   If rst303.EOF = False Then
   	SmartTags("ID_OP_4") = rst303.Fields(0).Value
   	SmartTags("Name_OP_4") = rst303.Fields(1).Value
   	rst303.MoveNext
   Else
   	SmartTags("ID_OP_4") = 0
   	SmartTags("Name_OP_4") = "Vacio"
   End If
   
   If rst303.EOF = False Then
   	SmartTags("ID_OP_5") = rst303.Fields(0).Value
   	SmartTags("Name_OP_5") = rst303.Fields(1).Value
   	rst303.MoveNext
   Else
   	SmartTags("ID_OP_5") = 0
   	SmartTags("Name_OP_5") = "Vacio"
   End If
   
   rst303.close
   conn303.close
   
   Set rst303 = Nothing
   Set conn303 = Nothing

VB script "S20_Generador_Inf"
   Dim NombreInf_Pl, NombreInf_Lavs
   
   'Informe de planchadoras
   bfde4b54-0db7-4817-8032-87127bf19bb9 "Se llamo a S07"
   NombreInf_Pl = S07_InformeDiario_Planchas()
   bfde4b54-0db7-4817-8032-87127bf19bb9 "Se Salio de S07"
   
   ' Informe unico de lavadoras
   bfde4b54-0db7-4817-8032-87127bf19bb9 "Se llamo a S23"
   NombreInf_Lavs = S23_Creador_InformeDiarioLavs_Gral()
   bfde4b54-0db7-4817-8032-87127bf19bb9 "Se Salio de S23"
   
   Call S30_EnvioInformes_Email(NombreInf_Pl, NombreInf_Lavs)

VB script "S30_EnvioInformes_Email"
   '## ENVIAR INFORME POR EMAIL
   
   Dim appOutlook 'As OUTLOOK.APPLICATION
   Dim mlNewMail 'As MailItem
   Dim objEntry
   Dim Text
   
   Const addressee = "crj@eprocsrl.com.ar; danielst@live.com.ar; josemariacullen@hotmail.com;"' zekeserio@hotmail.com;"
   
   ' Text to be sent 
   
   Text = "Informe diario"
   
   Set appOutlook = CreateObject("OUTLOOK.APPLICATION")
   
   
   'Generating and sending an e-mail:
   Set mlNewMail = appOutlook.CreateItem(0)
   mlNewMail.Display
   mlNewMail.To = addressee
   mlNewMail.Subject = "Informe Diario de produccion"
   
   
   If InStr(Arch1,"ERR") <> 0 Then
   	Text = Text + vbCrLf +_
   	"Error al Crear el informe de Planchadoras"
   Else
   	mlNewMail.Attachments.Add CStr(Arch1)
   End If
   
   If InStr(Arch2,"ERR") <> 0 Then
   	Text = Text + vbCrLf +_
   	"Error al Crear el informe de Lavadoras"
   Else
   	mlNewMail.Attachments.Add CStr(Arch2)
   End If
   
   
   mlNewMail.Body = Text
   mlNewMail.save
   mlNewMail.send 
   
   'Error routine
   If Err.Number <> 0 Then
   	bfde4b54-0db7-4817-8032-87127bf19bb9 "Error al enviar el email #" & Err.Number & " " & Err.Description
   End If

VB script "S304_ActualizarOpEnPrincipal"
   'Declaracion de Variables locales
   Dim conn21, rst21, Consulta
   
   On Error Resume Next
   
   Set conn21 = CreateObject("ADODB.Connection")
   Set rst21 = CreateObject("ADODB.Recordset")
   
   'Abrir BDD
   conn21.Open "Provider=MSDASQL;Initial Catalog=Lavadero;DSN=Lavadero"
   
   
   'Chequeo de error
   If Err.Number <> 0 Then
   	bfde4b54-0db7-4817-8032-87127bf19bb9 "Error #" & Err.Number & " " & Err.Description
   	Err.Clear 
   	Set conn21 = Nothing
   	Exit Sub
   End If
   
   If LavNro = 1 Then	
   	
   	Consulta = "SELECT * FROM Op_Lavadoras WHERE  ID = '" & SmartTags("Lav1_Operador") &"';"
   	
   	'Ejecutar consulta
   	Set rst21 = conn21.Execute(Consulta)
   
   	SmartTags("Lav1_Operador_Str")= rst21.Fields(1).Value
   	
   End If
   
   If LavNro = 2 Then	
   	Consulta = "SELECT * FROM Op_Lavadoras WHERE  ID = '" & SmartTags("Lav2_Operador") &"';"
   	
   	'Ejecutar consulta
   	Set rst21 = conn21.Execute(Consulta)
   
   	SmartTags("Lav2_Operador_Str")= rst21.Fields(1).Value
   	
   End If
   
   If LavNro = 3 Then	
   	Consulta = "SELECT * FROM Op_Lavadoras WHERE  ID = '" & SmartTags("Lav3_Operador") &"';"
   	
   	'Ejecutar consulta
   	Set rst21 = conn21.Execute(Consulta)
   
   	SmartTags("Lav3_Operador_Str")= rst21.Fields(1).Value
   	
   End If
   
   If LavNro = 4 Then	
   	Consulta = "SELECT * FROM Op_Lavadoras WHERE  ID = '" & SmartTags("Lav4_Operador") &"';"
   	
   	'Ejecutar consulta
   	Set rst21 = conn21.Execute(Consulta)
   
   	SmartTags("Lav4_Operador_Str")= rst21.Fields(1).Value
   	
   End If
   
   
   rst21.close 
   
   conn21.close
   
   Set rst21 = Nothing
   Set conn21 = Nothing

VB script "SA1_email_Vibr"
   	
   	
   	Dim appOutlook 'As OUTLOOK.APPLICATION
   	Dim mlNewMail 'As MailItem
   	Dim objEntry
   	Dim Text, cliente_0, cliente_1, cliente_2, operario, carga, programa
   	Dim cliente_0_str, cliente_1_str, cliente_2_str, operario_str
   		
   	Const addressee = "crj@eprocsrl.com.ar; danielst@live.com.ar;"' josemariacullen@hotmail.com; zekeserio@hotmail.com;"	
   	
   	
   ' ######### Consulta para obtener el listado actualizado de clientes ############
   	Dim conncli, rstcli , ConsultaCli
   	
   	Set conncli = CreateObject("ADODB.Connection")
   	Set rstcli = CreateObject("ADODB.Recordset")
   	
   	'Open data source - Datenquelle öffnen
   	conncli.Open "Provider=MSDASQL;Initial Catalog=Lavadero;DSN=Lavadero"
   	'Error routine - Fehlerroutine
   	If Err.Number <> 0 Then
   		bfde4b54-0db7-4817-8032-87127bf19bb9 "Conexion Error a Cli_Lavadoras#" & Err.Number & " " & Err.Description
   		Err.Clear
   		Set conncli = Nothing  
   		Exit Sub
   	End If
   	
   	ConsultaCli = "SELECT * FROM Cli_Lavadoras;"
   	
   	'Ejecutar consulta
   	Set rstcli = conncli.Execute(ConsultaCli)
   '''''''''''''''''''''''''''''''''''''''''''''''''''''''''''''''''''''''
   
   	
   ' ######### Consulta para obtener el listado actualizado de OPERADORES ############
   Dim connope, rstope , Consultaope
   
   Set connope = CreateObject("ADODB.Connection")
   Set rstope = CreateObject("ADODB.Recordset")
   
   'Open data source - Datenquelle öffnen
   connope.Open "Provider=MSDASQL;Initial Catalog=Lavadero;DSN=Lavadero"
   'Error routine - Fehlerroutine
   If Err.Number <> 0 Then
   	bfde4b54-0db7-4817-8032-87127bf19bb9 "Conexion Error a Op_Lavadoras" & Err.Number & " " & Err.Description
   	Err.Clear
   	Set connope = Nothing  
   	Exit Sub
   End If
   
   Consultaope = "SELECT * FROM Op_Lavadoras;"
   
   'Ejecutar consulta
   Set rstope = connope.Execute(Consultaope)
   ''''''''''''''''''''''''''''''''''''''''''''''''''''''''''''''''''''''''''''''''
   	
   '## ENVIAR Aviso POR EMAIL AVISO FALLA VIBRACION LAVADORA 1
   
   If  SmartTags("Lav1_AlarmaVibracion") = True Then
   
   	cliente_0 = SmartTags("Lav1_Cliente_0")
   	cliente_1 = SmartTags("Lav1_Cliente_1")
   	cliente_2 = SmartTags("Lav1_Cliente_2")
   		
   	operario = SmartTags("Lav1_Operador")
   	
   	carga = SmartTags("Lav1_CantRopa")
   	
   	programa =  S12_Conversor_BCD_to_Int(SmartTags("Lav1_Programa"))
   	
   
   	' Establecer los clientes
   	Do While rstcli.EOF = False
   		If (rstcli.Fields(0).Value = cliente_0) Then 
   			cliente_0_str = Trim(rstcli.Fields(1).Value)
   		End If
   
   		If (rstcli.Fields(0).Value = cliente_1) Then 
   			cliente_1_str = Trim(rstcli.Fields(1).Value)
   		End If
   
   		If (rstcli.Fields(0).Value = cliente_2) Then 
   			cliente_2_str = Trim(rstcli.Fields(1).Value)
   		End If
   			
   		rstcli.MoveNext
   	Loop
   	
   	' Establecer operador
   	Do While rstope.EOF = False
   		If (rstope.Fields(0).Value = operario) Then 
   			operario_str = Trim(rstope.Fields(1).Value)
   		End If	
   		rstope.MoveNext
   	Loop
   		
   	' Text to be sent 
   	
   	Text = "AVISO DE FALLA POR VIBRACION EN LAVADORA 1" + vbCrLf +_
   			"Hora: " + CStr(Date()) + " " + CStr(Time()) + vbCrLf +_
   			"Clientes: " + cliente_0_str + "/" + cliente_1_str + "/" + cliente_2_str + vbCrLf +_
   			"Operario: " + operario_str + vbCrLf +_
   			"Carga: " + CStr(carga/10) + " Kg" + vbCrLf +_
   			"Programa: " + CStr(programa)
   	
   	Set appOutlook = CreateObject("OUTLOOK.APPLICATION")
   	
   	
   	'Generating and sending an e-mail:
   	Set mlNewMail = appOutlook.CreateItem(0)
   	mlNewMail.Display
   	mlNewMail.To = addressee
   	mlNewMail.Subject = "Aviso de falla por vibracion en lavadora 1"
   	mlNewMail.Body = Text
   	mlNewMail.save
   	mlNewMail.send 
   	
   End If
   
   '## ENVIAR Aviso POR EMAIL AVISO FALLA VIBRACION LAVADORA 2
   
   If  SmartTags("Lav2_AlarmaVibracion") = True Then
   
   	cliente_0 = SmartTags("Lav2_Cliente_0")
   	cliente_1 = SmartTags("Lav2_Cliente_1")
   	cliente_2 = SmartTags("Lav2_Cliente_2")
   		
   	operario = SmartTags("Lav2_Operador")
   	
   	carga = SmartTags("Lav2_CantRopa")
   	
   	programa =  S12_Conversor_BCD_to_Int(SmartTags("Lav2_Programa"))
   	
   
   	' Establecer los clientes
   	Do While rstcli.EOF = False
   		If (rstcli.Fields(0).Value = cliente_0) Then 
   			cliente_0_str = Trim(rstcli.Fields(1).Value)
   		End If
   
   		If (rstcli.Fields(0).Value = cliente_1) Then 
   			cliente_1_str = Trim(rstcli.Fields(1).Value)
   		End If
   
   		If (rstcli.Fields(0).Value = cliente_2) Then 
   			cliente_2_str = Trim(rstcli.Fields(1).Value)
   		End If
   			
   		rstcli.MoveNext
   	Loop
   	
   	' Establecer operador
   	Do While rstope.EOF = False
   		If (rstope.Fields(0).Value = operario) Then 
   			operario_str = Trim(rstope.Fields(1).Value)
   		End If	
   		rstope.MoveNext
   	Loop
   		
   	' Text to be sent 
   	
   	Text = "AVISO DE FALLA POR VIBRACION EN LAVADORA 2" + vbCrLf +_
   			"Hora: " + CStr(Date()) + " " + CStr(Time()) + vbCrLf +_
   			"Clientes: " + cliente_0_str + "/" + cliente_1_str + "/" + cliente_2_str + vbCrLf +_
   			"Operario: " + operario_str + vbCrLf +_
   			"Carga: " + CStr(carga/10) + " Kg" + vbCrLf +_
   			"Programa: " + CStr(programa)
   	
   	Set appOutlook = CreateObject("OUTLOOK.APPLICATION")
   	
   	
   	'Generating and sending an e-mail:
   	Set mlNewMail = appOutlook.CreateItem(0)
   	mlNewMail.Display
   	mlNewMail.To = addressee
   	mlNewMail.Subject = "Aviso de falla por vibracion en lavadora 2"
   	mlNewMail.Body = Text
   	mlNewMail.save
   	mlNewMail.send 
   	
   End If
   
   '## ENVIAR Aviso POR EMAIL AVISO FALLA VIBRACION LAVADORA 3
   
   If  SmartTags("Lav3_AlarmaVibracion") = True Then
   
   	cliente_0 = SmartTags("Lav3_Cliente_0")
   	cliente_1 = SmartTags("Lav3_Cliente_1")
   	cliente_2 = SmartTags("Lav3_Cliente_2")
   		
   	operario = SmartTags("Lav3_Operador")
   	
   	carga = SmartTags("Lav3_CantRopa")
   	
   	programa =  S12_Conversor_BCD_to_Int(SmartTags("Lav3_Programa"))
   	
   
   	' Establecer los clientes
   	Do While rstcli.EOF = False
   		If (rstcli.Fields(0).Value = cliente_0) Then 
   			cliente_0_str = Trim(rstcli.Fields(1).Value)
   		End If
   
   		If (rstcli.Fields(0).Value = cliente_1) Then 
   			cliente_1_str = Trim(rstcli.Fields(1).Value)
   		End If
   
   		If (rstcli.Fields(0).Value = cliente_2) Then 
   			cliente_2_str = Trim(rstcli.Fields(1).Value)
   		End If
   			
   		rstcli.MoveNext
   	Loop
   	
   	' Establecer operador
   	Do While rstope.EOF = False
   		If (rstope.Fields(0).Value = operario) Then 
   			operario_str = Trim(rstope.Fields(1).Value)
   		End If	
   		rstope.MoveNext
   	Loop
   		
   	' Text to be sent 
   	
   	Text = "AVISO DE FALLA POR VIBRACION EN LAVADORA 3" + vbCrLf +_
   			"Hora: " + CStr(Date()) + " " + CStr(Time()) + vbCrLf +_
   			"Clientes: " + cliente_0_str + "/" + cliente_1_str + "/" + cliente_2_str + vbCrLf +_
   			"Operario: " + operario_str + vbCrLf +_
   			"Carga: " + CStr(carga/10) + " Kg" + vbCrLf +_
   			"Programa: " + CStr(programa)
   	
   	Set appOutlook = CreateObject("OUTLOOK.APPLICATION")
   	
   	
   	'Generating and sending an e-mail:
   	Set mlNewMail = appOutlook.CreateItem(0)
   	mlNewMail.Display
   	mlNewMail.To = addressee
   	mlNewMail.Subject = "Aviso de falla por vibracion en lavadora 3"
   	mlNewMail.Body = Text
   	mlNewMail.save
   	mlNewMail.send 
   	
   End If
   
   
   '## ENVIAR Aviso POR EMAIL AVISO FALLA VIBRACION LAVADORA 3
   
   If  SmartTags("Lav4_AlarmaVibracion") = True Then
   
   	cliente_0 = SmartTags("Lav4_Cliente_0")
   	cliente_1 = SmartTags("Lav4_Cliente_1")
   	cliente_2 = SmartTags("Lav4_Cliente_2")
   		
   	operario = SmartTags("Lav4_Operador")
   	
   	carga = SmartTags("Lav4_CantRopa")
   	
   	programa =  S12_Conversor_BCD_to_Int(SmartTags("Lav4_Programa"))
   	
   
   	' Establecer los clientes
   	Do While rstcli.EOF = False
   		If (rstcli.Fields(0).Value = cliente_0) Then 
   			cliente_0_str = Trim(rstcli.Fields(1).Value)
   		End If
   
   		If (rstcli.Fields(0).Value = cliente_1) Then 
   			cliente_1_str = Trim(rstcli.Fields(1).Value)
   		End If
   
   		If (rstcli.Fields(0).Value = cliente_2) Then 
   			cliente_2_str = Trim(rstcli.Fields(1).Value)
   		End If
   			
   		rstcli.MoveNext
   	Loop
   	
   	' Establecer operador
   	Do While rstope.EOF = False
   		If (rstope.Fields(0).Value = operario) Then 
   			operario_str = Trim(rstope.Fields(1).Value)
   		End If	
   		rstope.MoveNext
   	Loop
   		
   	' Text to be sent 
   	
   	Text = "AVISO DE FALLA POR VIBRACION EN LAVADORA 4" + vbCrLf +_
   			"Hora: " + CStr(Date()) + " " + CStr(Time()) + vbCrLf +_
   			"Clientes: " + cliente_0_str + "/" + cliente_1_str + "/" + cliente_2_str + vbCrLf +_
   			"Operario: " + operario_str + vbCrLf +_
   			"Carga: " + CStr(carga/10) + " Kg" + vbCrLf +_
   			"Programa: " + CStr(programa)
   	
   	Set appOutlook = CreateObject("OUTLOOK.APPLICATION")
   	
   	
   	'Generating and sending an e-mail:
   	Set mlNewMail = appOutlook.CreateItem(0)
   	mlNewMail.Display
   	mlNewMail.To = addressee
   	mlNewMail.Subject = "Aviso de falla por vibracion en lavadora 4"
   	mlNewMail.Body = Text
   	mlNewMail.save
   	mlNewMail.send 
   	
   End If
   
   
   
   '########################################################################
   'Close data source - Datenquelle schließen
   
   conncli.close
   Set rstcli = Nothing
   Set conncli = Nothing
   
   connope.close
   Set rstope = Nothing
   Set connope = Nothing

VB script "S23_Creador_InformeDiarioLavs_Gral"
   S23_Creador_InformeDiarioLavs_Gral = "ERROR"
   
   If Err.Number <> 0 Then
   	bfde4b54-0db7-4817-8032-87127bf19bb9 "Erorr anterior a  'S23_Creador_InformeDiarioLavs_Gral' #" & Err.Number & " " & Err.Description
   	Err.Clear
   End If
   
   bfde4b54-0db7-4817-8032-87127bf19bb9 "Entro a S23"
   'Declaration of local tags 
   
   Dim cantidadDeRegistros
   	cantidadDeRegistros = 60
   Dim cantidadDeLavadoras
   	cantidadDeLavadoras = 4
   
   Dim conn, rst, i, j, indicehoja, k, l
   
   Dim Consulta
   Dim conncli, rstcli , ConsultaCli
   Dim connope, rstope , Consultaope
   Dim connfall,rstfall, Consultafall
   
   Dim DiaAnterior
   Dim horaInicioDia, horaFinDia
   Dim tcargaLav(4), tciclosLav(4), tciclosnvLav(4)
   Dim HoraFin, HoraInicio
   Dim thoras , tcarga, tciclos, thorasdate, thorasSdate(4), thorasmuertodate
   Dim rst2
   
   ' Creo Variables locales para poder iterar con los datos
   Dim VarCLINro_0(60), 	VarCLINro_1(60)
   Dim VarCLINro_2(60), 	VarC(60)
   Dim VarPR(60), 		VarHI(60)
   Dim VarHF(60), 		VarOPNro(60)
   Dim VarNV(60), 		VarEsp(60)
   Dim VarCLIStr(60), 	VarOPStr(60)
   Dim band_1(60), 	VarHE(60)
   Dim VarCicloOk(60), VarFalla(60), VarCicloOkAns(60)
   Dim VarCicloOk_CN(60)
   Dim VarFallaStr(60), VarFallaSQL(60)
   Dim LavadoraNro
   Dim indexMuertoFin(4),indexMuerto(4)
   Dim inicioderegistrosdelavadora
   Dim Programas(15), p, Promedio(4), PromedioTotal, Programas_Lav4(15)
   Dim fin
   Dim tiemponulo , thorasAns, tdias
   Dim lavEnFalla
   
   'Inicializacion Global de variables
   For p = 1 To 15
   	Programas(p) = 0
   	Programas_Lav4(p) = 0
   Next
   '
   If Err.Number <> 0 Then
   	bfde4b54-0db7-4817-8032-87127bf19bb9 "Consulta Lav Error 1#" & Err.Number & " " & Err.Description
   	Err.Clear
   	'Close data source	
   	Set conn = Nothing
   	Set rst = Nothing 
   	
   	Exit Function
   End If
   
   tiemponulo = FormatDateTime("2020-02-05 00:00:00", 4)
   
   For i = 1 To cantidadDeRegistros
   	VarNV(i) 		= 0
   	VarHI(i) 		= FormatDateTime("2020-02-05 00:00:00", 4)
   	VarHF(i) 		= FormatDateTime("2020-02-05 00:00:00", 4)
   	VarHE(i) 		= FormatDateTime("2020-02-05 00:00:00", 4)		
   	VarCLIStr(i) 	= "                                       "
   	VarOPStr(i) 	= "                                       "
   	band_1(i)		= 0
   	VarCicloOk(i)	= "X" ' negativo "O"; positivo "P"
   	VarFalla(i)		= 0
   	VarFallaStr(i)	= "                                       "	
   Next
   
   
   
   If Err.Number <> 0 Then
   	bfde4b54-0db7-4817-8032-87127bf19bb9 "Consulta Lav Error 2#" & Err.Number & " " & Err.Description
   	Err.Clear
   	'Close data source
   	Set conn = Nothing
   	Set rst = Nothing 
   	
   	Exit Function
   End If
   
   thoras = FormatDateTime("2020-02-05 00:00:00", 4)
   
   indicehoja = 1
   
   'DiaAnterior = Date() ' Es el día actual
   'DiaAnterior = DateAdd("d",-1, DiaAnterior)
   DiaAnterior = FormatDateTime(CStr(SmartTags("Ver_DIA_X")), 2)
   
   
   If Err.Number <> 0 Then
   	bfde4b54-0db7-4817-8032-87127bf19bb9 "Consulta Lav Error 3#" & Err.Number & " " & Err.Description
   	Err.Clear
   	'Close data source
   	Set conn = Nothing
   	Set rst = Nothing 
   	Exit Function
   End If
   
   
   For i = 1 To cantidadDeLavadoras
   	tcargaLav(i)		= 0
   	tciclosLav(i)		= 0
   	tciclosnvLav(i) 	= 0
   
   	Promedio(i)			= 0
   Next
   
   If Err.Number <> 0 Then
   	bfde4b54-0db7-4817-8032-87127bf19bb9 "Consulta Lav Error 5#" & Err.Number & " " & Err.Description
   	Err.Clear
   	'Close data source
   	Set conn = Nothing
   	Set rst = Nothing 
   	
   	Exit Function
   End If
   
   tcarga 			= 0
   tciclos 		= 0
   lavEnFalla		= 1
   
   'Analisar si hay error e imprimirlo
   If Err.Number <> 0 Then
   	bfde4b54-0db7-4817-8032-87127bf19bb9 "Consulta Lav Error 6#" & Err.Number & " " & Err.Description
   	Err.Clear
   	'Close data source
   	Set conn = Nothing
   	Set rst = Nothing 
   	
   	Exit Function
   End If
   
   ' Comienzo de procesamiento de datos
   On Error Resume Next
   
   For LavadoraNro = 1 To cantidadDeLavadoras
   	'""""""""""""""""""""""""""""""""""""""""""""""""""""""""""""""""""""""""""""""""""""
   	' #################   Generacion de consulta a BDD Lavadora   ######################
   	'------------------------------------------------------------------------------------
   	'############ Estructura de datos de la Tabla Lav1 #################################
   	
   	'0			1			2			3			4			5			6			7			8			
   	'|FechaFin	|FechIni	|Cliente_0	|Cliente_1	|Cliente_2	|Operario	|Carga		|Programa	|Valido
   	'|Date		|Date		|Int		|Int		|Int		|Int		|Int 100g	|Int		|Bool
   	
   	'##################################################################################
   		
   	'''''''''''''''''''''''''''''''''''''''''''''''''''''''''''''''''''''''''''''
   	' #################   Procesamieno de Datos   #############################
   	'----------------------------------------------------------------------------
   	
   	'Ejecutar consulta
   	
   	Consulta = "SELECT * FROM Lav" & LavadoraNro & " WHERE cast(fechafin As Date) = '"
   	Consulta = Consulta & CStr(Year(DiaAnterior)) & "-" & CStr(Month(DiaAnterior)) & "-" & CStr(Day(DiaAnterior)) & "' "
   	Consulta = Consulta & " order by fechafin"
   	
   	Set conn = CreateObject("ADODB.Connection")
   	conn.Open "Provider=MSDASQL;Initial Catalog=Lavadero;DSN=Lavadero"
   	Set rst2 = CreateObject("ADODB.Recordset")
   	Set rst2 = conn.Execute(Consulta)	
   	
   	inicioderegistrosdelavadora = indicehoja
   	i = indicehoja
   	
   	'ShowSystemAlarm "Entra al loop de Lectura de registros de Lav nro " & LavadoraNro
   	
   	Do While rst2.EOF = False
   			
   		VarCLINro_0(i) 	= rst2.Fields(2).Value
   		VarCLINro_1(i) 	= rst2.Fields(3).Value
   		VarCLINro_2(i) 	= rst2.Fields(4).Value
   		VarC(i) 		= rst2.Fields(6).Value / 10
   		VarPR(i) 		= rst2.Fields(7).Value
   		VarHI(i) 		= FormatDateTime(CStr(rst2.Fields(1).Value), 4) 'Devuelve la parte Time de la fecha
   		VarHF(i) 		= FormatDateTime(CStr(rst2.Fields(0).Value), 4)
   		VarOPNro(i)		= rst2.Fields(5).Value
   		VarNV(i) 		= 1	
   		VarCicloOk_CN(i)= rst2.Fields(9).Value
   		
   		If rst2.Fields(8).Value = 0 Then ' Si el ciclo es no valido
   			If VarCicloOk_CN(i) = 0 Then
   				VarCicloOk(i) 			= "O" ' negativo "O"; positivo "P"
   			Else
   				VarCicloOk(i) 			= "8" ' negativo "O"; positivo "P"
   			End If
   			tciclosnvLav(LavadoraNro) = tciclosnvLav(LavadoraNro) +1
   		Else
   			VarCicloOk(i) 			= "P" ' negativo "O"; positivo "P"
   			If VarPR(i) <> 12 And VarPR(i) <> 11 Then
   				tciclosLav(LavadoraNro) = tciclosLav(LavadoraNro) 	+ 1
   			End If
   			'tcargaLav(LavadoraNro)	= tcargaLav(LavadoraNro) 	+ VarC(i)
   				
   				' Suma de formulas utilizadas
   			If LavadoraNro <> 4 Then
   				Programas(VarPR(i)) = Programas(VarPR(i)) + 1
   			Else
   				Programas_Lav4(VarPR(i)) = Programas_Lav4(VarPR(i)) + 1
   			End If
   			
   		End If
   		
   		'Suma de Carga lavada
   		If i > 1 Then
   			If VarCicloOk(i) = "P" And VarPR(i) <> 12 And VarPR(i) <> 11 Or (VarCicloOkAns(i) = "O" And (VarPR(i) = 12 Or VarPR(i) = 11)) Then
   				tcargaLav(LavadoraNro)	= tcargaLav(LavadoraNro) 	+ VarC(i)
   			End If
   		Else
   			If VarCicloOk(i) = "P" And VarPR(i) <> 12 And VarPR(i) <> 11 Then
   				tcargaLav(LavadoraNro)	= tcargaLav(LavadoraNro) 	+ VarC(i)
   			End If
   		End If
   		
   	
   		'Calculo de tiempo muerto si corresponde
   		If i > 1 Then'VarHI(i-1) <> tiemponulo Then
   			VarHE(i-1) = DateAdd("h", Hour(VarHI(i)) - Hour(VarHF(i-1)), VarHE(i-1))
   			VarHE(i-1) = DateAdd("n", Minute(VarHI(i)) - Minute(VarHF(i-1)), VarHE(i-1))				
   			VarHE(i-1) = DateAdd("s", Second(VarHI(i)) - Second(VarHF(i-1)), VarHE(i-1))
   		End If
   		
   		thoras = DateAdd("h", Hour(VarHF(i)) - Hour(VarHI(i)), thoras)
   		thoras = DateAdd("n", Minute(VarHF(i)) - Minute(VarHI(i)), thoras)
   		thoras = DateAdd("s", Second(VarHF(i)) - Second(VarHI(i)), thoras)
   		
   		If Hour(thoras) < Hour(thorasAns) Then
   			tdias = tdias + 1 
   			thorasAns = thoras
   		Else
   			thorasAns = thoras
   		End If
   		
   		If i > 1 Then
   			VarCicloOkAns(i) = VarCicloOk(i)
   		End If
   		
   		'Indice de lavados		
   		i = i + 1
   		
   		
   		rst2.MoveNext
   		
   		If Err.Number <> 0 Then
   			bfde4b54-0db7-4817-8032-87127bf19bb9 "Error en la asignacion de variables locales en loop#" & Err.Number & " " & Err.Description
   			Err.Clear
   			Set conn = Nothing  
   			Exit Function
   		End If
   	Loop
   	
   	'ShowSystemAlarm "Sale del loop de Lectura de registros de Lav nro " & LavadoraNro
   	
   	If Err.Number <> 0 Then
   		bfde4b54-0db7-4817-8032-87127bf19bb9 "Error en la asignacion de variables locales luego del loop#" & Err.Number & " " & Err.Description
   		Err.Clear
   		Set conn = Nothing  
   		Exit Function
   	End If
   	
   	VarCicloOk(i) 	= "P" ' negativo "O"; positivo "P"
   	VarC(i) 		= tcargaLav(LavadoraNro)
   	VarNV(i) 		= 1
   	
   	'''	
   	VarCLIStr		(i)	= "Total Lav Maq " & CStr(LavadoraNro)
   	VarPR			(i)	= 0
   	VarHI			(i)	= 0	
   	VarHF			(i)	= 0
   	VarOPStr		(i) = " "
   	VarFallaStr		(i)	= " "
   	VarHE			(i) = 0
   	''''
   	indicehoja = i + 1
   	
   	'Indice para sumar tiempos muertos
   	indexMuertoFin(LavadoraNro) 	= i - 1
   	indexMuerto(LavadoraNro)		= i - 2
   	SmartTags("BCDtoInt")			= indexMuerto(LavadoraNro)
   	SmartTags("BCDtoInt_Entrada")	= inicioderegistrosdelavadora
   	
   	'Calculo de tiempos muertos parciales de lavadoras
   	k = inicioderegistrosdelavadora
   
   	fin = False
   	
   	'ShowSystemAlarm "Entra al loop de suma de tiempos muertos de lav  " & LavadoraNro
   		
   	Do While fin = False
   		VarHE(indexMuertoFin(LavadoraNro)) = DateAdd("h",Hour(VarHE(k)), VarHE(indexMuertoFin(LavadoraNro)))
   		VarHE(indexMuertoFin(LavadoraNro)) = DateAdd("n",Minute(VarHE(k)), VarHE(indexMuertoFin(LavadoraNro)))			
   		VarHE(indexMuertoFin(LavadoraNro)) = DateAdd("s",Second(VarHE(k)), VarHE(indexMuertoFin(LavadoraNro)))
   		
   		If (k < indexMuerto(LavadoraNro)) Then
   			k = k + 1
   		Else
   			fin = True
   		End If
   	Loop
   	
   	'ShowSystemAlarm "Sale del loop de suma de tiempos muertos de lav  " & LavadoraNro
   	
   	If Err.Number <> 0 Then
   		bfde4b54-0db7-4817-8032-87127bf19bb9 "Error en la asignacion de variables locales a lo ultimo#" & Err.Number & " " & Err.Description
   		Err.Clear
   		Set conn = Nothing  
   		Exit Function
   	End If
   	
   	
   	conn.close
   	Set rst2 = Nothing
   	Set conn = Nothing
   	
   Next
   
   'ShowSystemAlarm "Sale del loop general de rst"
   
   'Armado de tiempo total de lavado
   Dim tHorasString
   tHorasString = SA2_TotalTimeToString(tdias, thoras)
   
   'calculo de tiempo muerto total y promedios de las 4 lavadoras
   Dim indiceFinal
   indiceFinal = indexMuertoFin(4) +2
   'ShowSystemAlarm "entra loop Promedio, Var E"
   For k = 1 To 4
   	
   	VarHE(indiceFinal) = DateAdd("h",Hour(VarHE(indexMuertoFin(k))), VarHE(indiceFinal))
   	VarHE(indiceFinal) = DateAdd("n",Minute(VarHE(indexMuertoFin(k))), VarHE(indiceFinal))				
   	VarHE(indiceFinal) = DateAdd("s",Second(VarHE(indexMuertoFin(k))), VarHE(indiceFinal))
   	
   	If tciclosLav(k) <> 0 Then
   		Promedio(k) = tcargaLav(k) / tciclosLav(k)	
   	End If
   Next
   'ShowSystemAlarm "Sale loop Promedio, Var E"
   
   VarNV			(indiceFinal) 	= 1
   	
   If Err.Number <> 0 Then
   	bfde4b54-0db7-4817-8032-87127bf19bb9 "Error en la asignacion de variables generales 1#" & Err.Number & " " & Err.Description
   	Err.Clear
   	Set conn = Nothing  
   	Exit Function
   End If
   
   '###################################3###################################################
   '####### AHORA SE COPIAN LOS REGISTROS EN LAS VARIABLES DE LAS TABLAS   ################
   '###################################3###################################################
   
   ' ######### Consulta para obtener el listado actualizado de clientes ############
   
   Set conncli = CreateObject("ADODB.Connection")
   Set rstcli = CreateObject("ADODB.Recordset")
   
   'Open data source - Datenquelle öffnen
   conncli.Open "Provider=MSDASQL;Initial Catalog=Lavadero;DSN=Lavadero"
   'Error routine - Fehlerroutine
   If Err.Number <> 0 Then
   	bfde4b54-0db7-4817-8032-87127bf19bb9 "Conexion Error a Cli_Lavadoras#" & Err.Number & " " & Err.Description
   	Err.Clear
   	Set conncli = Nothing  
   	Exit Function
   End If
   
   ConsultaCli = "SELECT * FROM Cli_Lavadoras;"
   
   'Ejecutar consulta
   Set rstcli = conncli.Execute(ConsultaCli)
   ''''''''''''''''''''''''''''''''''''''''''''''''''''''''''''''''''''''''''''''''
   
   ' ######### Consulta para obtener el listado actualizado de OPERADORES ############
   
   Set connope = CreateObject("ADODB.Connection")
   Set rstope = CreateObject("ADODB.Recordset")
   
   'Open data source - Datenquelle öffnen
   connope.Open "Provider=MSDASQL;Initial Catalog=Lavadero;DSN=Lavadero"
   'Error routine - Fehlerroutine
   If Err.Number <> 0 Then
   	bfde4b54-0db7-4817-8032-87127bf19bb9 "Conexion Error a Op_Lavadoras" & Err.Number & " " & Err.Description
   	Err.Clear
   	Set connope = Nothing  
   	Exit Function
   End If
   
   Consultaope = "SELECT * FROM Op_Lavadoras;"
   
   'Ejecutar consulta
   Set rstope = connope.Execute(Consultaope)
   ''''''''''''''''''''''''''''''''''''''''''''''''''''''''''''''''''''''''''''''''
   
   
   ' Establecer los clientes
   j = 1
   Do While rstcli.EOF = False
   	For j = 1 To cantidadDeRegistros 
   		If (rstcli.Fields(0).Value = VarCLINro_0(j)) Then ' Si el ciclo es no valido
   			If band_1(j) = 0 Then
   				VarCLIStr(j) = Trim(rstcli.Fields(1).Value)
   				band_1(j) = 1
   			Else
   				VarCLIStr(j) = VarCLIStr(j) + "/" + Trim(rstcli.Fields(1).Value)
   			End If
   		End If
   
   		If (rstcli.Fields(0).Value = VarCLINro_1(j)) Then ' Si el ciclo es no valido
   			If band_1(j) = 0 Then
   				VarCLIStr(j) = Trim(rstcli.Fields(1).Value)
   				band_1(j) = 1
   			Else
   				VarCLIStr(j) = VarCLIStr(j) + "/" + Trim(rstcli.Fields(1).Value)
   			End If
   		End If
   
   		If (rstcli.Fields(0).Value = VarCLINro_2(j)) Then ' Si el ciclo es no valido
   			If band_1(j) = 0 Then
   				VarCLIStr(j) = Trim(rstcli.Fields(1).Value)
   				band_1(j) = 1
   			Else
   				VarCLIStr(j) = VarCLIStr(j) + "/" + Trim(rstcli.Fields(1).Value)
   			End If
   		End If
   		
   	Next
   	rstcli.MoveNext
   Loop
   
   
   If Err.Number <> 0 Then
   	bfde4b54-0db7-4817-8032-87127bf19bb9 "Error en establecer los clientes#" & Err.Number & " " & Err.Description
   	Err.Clear
   	Set conncli = Nothing  
   	Exit Function
   End If
   
   ' Establecer los operarios
   j = 1
   Do While rstope.EOF = False
   	For j = 1 To cantidadDeRegistros
   		If (rstope.Fields(0).Value = VarOPNro(j)) Then ' Si el ciclo es no valido
   			VarOPStr(j) = Trim(rstope.Fields(1).Value)
   		End If
   	Next
   	rstope.MoveNext
   Loop
   
   If Err.Number <> 0 Then
   	bfde4b54-0db7-4817-8032-87127bf19bb9 "Error en establecer los operadores#" & Err.Number & " " & Err.Description
   	Err.Clear
   	Set connope = Nothing  
   	Exit Function
   End If
   
   '########################################################################
   'Close data source - Datenquelle schließen
   
   conncli.close
   Set rstcli = Nothing
   Set conncli = Nothing
   
   connope.close
   Set rstope = Nothing
   Set connope = Nothing
   
   ' Direccionamiento de variables locales a variables de salida
   tcarga =	tcargaLav(1) + tcargaLav(2) + tcargaLav(3) + tcargaLav(4)
   VarCLIStr		(indiceFinal)	= " "
   VarC			(indiceFinal)	= tcarga
   VarPR			(indiceFinal)	= 0
   VarHI			(indiceFinal)	= 0	
   VarHF			(indiceFinal)	= 0
   VarOPStr		(indiceFinal) 	= " "
   VarCicloOk		(indiceFinal) 	= "P" ' negativo "O"; positivo "P"
   VarFallaStr		(indiceFinal)	= " "
   	
   If Err.Number <> 0 Then
   	bfde4b54-0db7-4817-8032-87127bf19bb9 "Error variables vacias" & " Error#" & Err.Number & " " & Err.Description
   	Err.Clear
   	Exit Function
   End If
   
   'Direccionamiento tabla generales
   tciclos	=	tciclosLav(1) + tciclosLav(2) + tciclosLav(3)
   
   If Err.Number <> 0 Then
   	bfde4b54-0db7-4817-8032-87127bf19bb9 "Error Ciclos total" & " Error#" & Err.Number & " " & Err.Description
   	Err.Clear
   	Set conn = Nothing  
   	Exit Function
   End If
   
   If tciclos <> 0 Then
   	PromedioTotal 	= tcarga / tciclos
   End If
   
   If Err.Number <> 0 Then
   	bfde4b54-0db7-4817-8032-87127bf19bb9 "Error promedio6" & " Error#" & Err.Number & " " & Err.Description
   	Err.Clear
   	Set conn = Nothing  
   	Exit Function
   End If
   
   'Direccionamiento en tabla
   
   For i = 1 To cantidadDeRegistros
   	If VarNV(i) <> 1 Then
   		VarCLIStr		(i)		= ""
   		VarC			(i)		= 0
   		VarPR			(i)		= 0
   		VarHI			(i)		= 0
   		VarHF			(i)		= 0
   		VarOPStr		(i)		= ""
   		VarCicloOk		(i)		= "X"
   		VarFallaStr		(i)		= ""
   		VarHE			(i)		= 0
   	End If
   	
   	If Err.Number <> 0 Then
   		bfde4b54-0db7-4817-8032-87127bf19bb9 "Error en la carga de variables HMI, Indice #" & i & " Error#" & Err.Number & " " & Err.Description
   		Err.Clear
   		Set conn = Nothing  
   		Exit Function
   	End If
   Next
   
   bfde4b54-0db7-4817-8032-87127bf19bb9 "Salio de S23"
   
   '' %%%%%%%%%%%%%%%%%%%%%%%%%%%%%%%%%%%%%%%%%%%%%%%%%%%%%%%%%%%%%%%%%%%%%%%%%%%%%%%%%%%%%%%%%%%%%%%%%%%%%%%%%%%
   '' %%%%%%%%%%%%    IMPRESION DE DATOS EN INFORME    %%%%%%%%%%%%%%%%%%%%%%%%  XD  %%%%%%%%%%%%%%%%%%%%%%%%%%%%
   '' %%%%%%%%%%%%%%%%%%%%%%%%%%%%%%%%%%%%%%%%%%%%%%%%%%%%%%%%%%%%%%%%%%%%%%%%%%%%%%%%%%%%%%%%%%%%%%%%%%%%%%%%%%%
   
   Dim NameInfDiario
   
   NameInfDiario = "C:\ESPACIO DE TRABAJO\InformeDiario\" & "Lav" &(Replace(CStr(Date),"/","")& "-" &Replace(CStr(Time),":",""))&".xls"
   
   If Err.Number <> 0 Then
   	bfde4b54-0db7-4817-8032-87127bf19bb9 "Cambio de nombre Informe Diario Lavs 2 Error #" & Err.Number & " " & Err.Description
   	Err.Clear 
   	Exit Function
   End If
   
   ' Creacion devariables locales
   Dim objExcel
   Dim ColumnaMaquinado, ColumnaCantidades, ColumnaProm
   Dim objfso
   
   'Asignacion inicial de variables locales
   ColumnaMaquinado	= 12
   ColumnaCantidades	= 13
   ColumnaProm			= 14
   	
   'Creacion de Archivo .xls
   Set objExcel = CreateObject("Excel.Application")
   
   objExcel.Visible = False
   
   objExcel.Workbooks.Open "C:\ESPACIO DE TRABAJO\InformeDiario\Plantillas\InformeDiarioLavsExcelUnicoxls4_02.xls"
   'Fin creacion archivo .xls
   
   If Err.Number <> 0 Then
   	bfde4b54-0db7-4817-8032-87127bf19bb9 "NO SE ENCONTRO PLANILLA DE INFORMES LAVS GRAL" & Err.Number & " " & Err.Description
   	Err.Clear
   	Exit Function
   End If
   
   'Inserción de la fecha en el informe
   objExcel.Cells(2,6).Value = DiaAnterior
   
   Select Case Weekday(DiaAnterior)
   	Case 1		
   		objExcel.Cells(2,5).Value = "Domingo"
   	Case 2	
   		objExcel.Cells(2,5).Value = "Lunes"
   	Case 3	
   		objExcel.Cells(2,5).Value = "Martes"
   	Case 4	
   		objExcel.Cells(2,5).Value = "Miercoles"
   	Case 5	
   		objExcel.Cells(2,5).Value = "Jueves"
   	Case 6
   		objExcel.Cells(2,5).Value = "Viernes"
   	Case 7	
   		objExcel.Cells(2,5).Value = "Sabado"
   	Case Else
   		objExcel.Cells(2,5).Value = "Error"
   End Select
   
   ' Inserción de datos en el informe
   
   
   '$$$$$$$$$$$$$$$$$$$$$$ Fallas en el informe   $$$$$$$$$$$$$$$$$$$$$$
   
   Dim Fila, Columna
   
   '-----------------------------------
   'Insercion de fallas en informe
   
   Dim connf, rstf
   'Primero extraigo las fallas
   
   Set connf = CreateObject("ADODB.Connection")
   connf.Open "Provider=MSDASQL;Initial Catalog=Lavadero;DSN=Lavadero"
   Set rstf = CreateObject("ADODB.Recordset")
   
   	'Ejecutar consulta
   	
   	Consulta = "select * from LavAvisosFallas;"
   		
   	Set rstf = connf.Execute(Consulta)	
   	i = 1
   	Do While rstf.EOF = False
   		VarFallaSQL(i) = CStr(rstf.Fields(1).Value)
   		i = i + 1
   		rstf.MoveNext
   	Loop
   	
   	Set connf = Nothing  
   	Set rstf = Nothing
   
   '''Luego imprimo
   
   Fila = 34
   Columna = 12
   
   Set conn = CreateObject("ADODB.Connection")
   conn.Open "Provider=MSDASQL;Initial Catalog=Lavadero;DSN=Lavadero"
   Set rst2 = CreateObject("ADODB.Recordset")
   
   Dim lavNro, tmp_00, tmp_01, tmp_O, tmp_8
   
   	'Ejecutar consulta
   	
   	Consulta = "Select * from FallasLavs" &_
   		" where cast(fecha as Date) = '" &   CStr(Year(DiaAnterior)) & "-" & CStr(Month(DiaAnterior)) & "-" & CStr(Day(DiaAnterior)) & "' " &_
   		" And FallasLavs.falla <> '0';"
   		
   	Set rst2 = conn.Execute(Consulta)	
   		
   	Do While rst2.EOF = False
   		lavEnFalla = 1
   		'Impresion de falla al lado del ciclo
   		For i = 1 To cantidadDeRegistros
   			
   			
   			lavNro = rst2.Fields(2).Value
   			'ShowSystemAlarm "Lav Nro: #" & lavNro & ";LavenFalla: " & lavEnFalla
   			
   			tmp_O = InStr(CStr(VarCicloOk(i)),"O")
   			tmp_8 = InStr(CStr(VarCicloOk(i)),"8")
   			
   			'ShowSystemAlarm "tmp_O: #" & tmp_O & " Y tmp_8: #" & tmp_8
   			
   			If lavEnFalla = lavNro Then 
   				If tmp_O > 0 Or tmp_8 > 0 Then
   					'ShowSystemAlarm "Entro a super intermedio if #" & i
   					tmp_00 = FormatDateTime(CStr(rst2.Fields(1).Value), 4)
   					'ShowSystemAlarm "tmp_00 #" & tmp_00
   				
   					tmp_01 = VarHI(i)
   					'ShowSystemAlarm "tmp_01 #" & tmp_01
   					If tmp_01 < tmp_00 Then
   						tmp_01 = VarHF(i)
   						'ShowSystemAlarm "tmp_01_1 #" & tmp_01
   						If tmp_01 >= tmp_00 Then
   							VarFallaStr(i) = VarFallaSQL(rst2.Fields(3).Value)
   							'ShowSystemAlarm "Entro a super super if #" & i
   						End If
   						
   					End If
   				
   				End If
   				
   			End If
   			
   			If VarPR(i) = 0 Then 
   				'ShowSystemAlarm "Entro a if de lavEnFalla #" & i
   				lavEnFalla = lavEnFalla + 1
   			End If
   			
   			If Err.Number <> 0 Then
   				'ShowSystemAlarm "Error en bucle de registros#" & i & "#" & Err.Number & " " & Err.Description
   				Err.Clear
   			End If
   		Next
   			
   		If Fila > 1 And objExcel.Cells(Fila - 1,Columna + 1).Value <> CStr(rst2.Fields(1).Value) Then
   			objExcel.Cells(Fila,Columna).Value = CStr(rst2.Fields(2).Value)		
   			objExcel.Cells(Fila,Columna + 1).Value = CStr(rst2.Fields(1).Value)
   			objExcel.Cells(Fila,Columna + 2).Value = VarFallaSQL(rst2.Fields(3).Value)
   			Fila = Fila + 1
   		End If		
   		
   		If Err.Number <> 0 Then
   			'ShowSystemAlarm "bucle de fallas#" & Err.Number & " " & Err.Description
   			Err.Clear
   		End If
   		
   		rst2.MoveNext
   	Loop	
   	
   	Set rst2 = Nothing
   	
   	If Err.Number <> 0 Then
   		bfde4b54-0db7-4817-8032-87127bf19bb9 "Error en bucle de lavadoras#" & Err.Number & " " & Err.Description
   		Err.Clear
   	End If
   	
   	
   	'' Etiquetas de fallas
   	
   
   
   'Datos de Lavado generales
   
   'total de horas
   objExcel.Cells(2,10).Value	= tHorasString
   
   ' cantidades
   objExcel.Cells(26,ColumnaCantidades).Value	=	tcargaLav(1)
   objExcel.Cells(27,ColumnaCantidades).Value	=	tcargaLav(2)
   objExcel.Cells(28,ColumnaCantidades).Value	=	tcargaLav(3)
   
   objExcel.Cells(29,ColumnaCantidades).Value	=	(tcarga - tcargaLav(4))
   
   objExcel.Cells(26,ColumnaCantidades + 5).Value	=	tcargaLav(4)
   
   'Ciclos
   objExcel.Cells(26,ColumnaMaquinado).Value	=	tciclosLav(1)
   objExcel.Cells(27,ColumnaMaquinado).Value	=	tciclosLav(2)
   objExcel.Cells(28,ColumnaMaquinado).Value	=	tciclosLav(3)
   
   objExcel.Cells(29,ColumnaMaquinado).Value	=	tciclos
   
   objExcel.Cells(26,ColumnaMaquinado + 5).Value	=	tciclosLav(4)
   
   'Promedios
   objExcel.Cells(26,ColumnaProm).Value	=	Promedio(1)
   objExcel.Cells(27,ColumnaProm).Value	=	Promedio(2)
   objExcel.Cells(28,ColumnaProm).Value	=	Promedio(3)
   
   'objExcel.Cells(29,ColumnaProm).Value	=	PromedioTotal
   
   objExcel.Cells(26,ColumnaProm + 5).Value	=	Promedio(4)
   
   If Err.Number <> 0 Then
   	bfde4b54-0db7-4817-8032-87127bf19bb9 "Error en Impresion de datos generales" & Err.Number & " " & Err.Description
   	Err.Clear
   End If
   
   'Datos de cantidad de programas
   For i = 0 To 14
   	
   	If i <= 9 Then
   		objExcel.Cells(i+6,14).Value 	= Programas	(i + 1)
   	End If
   	
   	If i > 9 And i <= 11 Then
   		objExcel.Cells(i+11,14).Value	= Programas	(i + 1)
   	End If
   	
   	If i > 11 Then
   		objExcel.Cells(i+4,14).Value 	= Programas	(i + 1)
   	End If
   Next
   
   'Para lavadora 4
   For i = 0 To 14
   	
   	If i <= 9 Then
   		objExcel.Cells(i+6,19).Value 	= Programas_Lav4	(i + 1)
   	End If
   	
   	If i > 9 And i <= 11 Then
   		objExcel.Cells(i+11,19).Value	= Programas_Lav4	(i + 1)
   	End If
   	
   	If i > 11 Then
   		objExcel.Cells(i+4,19).Value 	= Programas_Lav4	(i + 1)
   	End If
   Next
   
   If Err.Number <> 0 Then
   	bfde4b54-0db7-4817-8032-87127bf19bb9 "Error en Impresion de formulas#" & Err.Number & " " & Err.Description
   	Err.Clear
   End If
   
   ' Direccionamiento de variables locales a variables de salida
   For i = 1 To cantidadDeRegistros
   	If VarCicloOk(i) <> "X" Then
   		If FormatDateTime(CStr(VarHI(i)), 4) <> FormatDateTime("2020-02-05 00:00:00", 4) Then
   	    	objExcel.Cells(i+4,1).Value = VarHI(i)
   	    End If
   	If Err.Number <> 0 Then
   		bfde4b54-0db7-4817-8032-87127bf19bb9 "Error en Impresion de datos en VarHI" & Err.Number & " " & Err.Description
   		Err.Clear
   	End If
   		If FormatDateTime(CStr(VarHF(i)), 4) <> FormatDateTime("2020-02-05 00:00:00", 4) Then
   	    	objExcel.Cells(i+4,2).Value = VarHF(i)
   	    End If
   	If Err.Number <> 0 Then
   		bfde4b54-0db7-4817-8032-87127bf19bb9 "Error en Impresion de datos en VarHF#"& Err.Number & " " & Err.Description
   		Err.Clear
   	End If
   	If VarC(i) <> 0 And VarCLIStr(i) <> " " And VarPR(i) <> 0 Then
   	    	objExcel.Cells(i+4,3).Value = VarHE(i)
   	End If
   	
   	If Err.Number <> 0 Then
   		bfde4b54-0db7-4817-8032-87127bf19bb9 "Error en Impresion de datos en VarHE#" & Err.Number & " " & Err.Description
   		Err.Clear
   	End If
   	
   	If VarC(i) <> 0 And VarCLIStr(i) = " " And VarPR(i) = 0 Then
   	    	objExcel.Cells(i+4,3).Value = VarHE(i)
   	    	objExcel.Cells(i+4,3).Font.Bold	= True
   	End If
   	
   	If Err.Number <> 0 Then
   		bfde4b54-0db7-4817-8032-87127bf19bb9 "Error en Impresion de datos en VarHE2#" & Err.Number & " " & Err.Description
   		Err.Clear
   	End If
   	
   	    If VarCLIStr(i) <> " " Then
   	    	objExcel.Cells(i+4,4).Value = VarCLIStr(i)
   		End If
   		
   	If Err.Number <> 0 Then
   		bfde4b54-0db7-4817-8032-87127bf19bb9 "Error en Impresion de datos en VarCLIStr#" & Err.Number & " " & Err.Description
   		Err.Clear
   	End If
   	
   		If VarCLIStr(i) <> " " And VarPR(i) = 0 Then
   			objExcel.Cells(i+4,4).Font.Bold = True
   			objExcel.Cells(i+4,6).Font.Bold = True
   		End If
   		
   	If Err.Number <> 0 Then
   		bfde4b54-0db7-4817-8032-87127bf19bb9 "Error en Impresion de datos en Bold#" & Err.Number & " " & Err.Description
   		Err.Clear
   	End If
   		
   		If VarPR(i) <> 0 Then
   	    	objExcel.Cells(i+4,5).Value = VarPR(i)
   		End If
   		
   	If Err.Number <> 0 Then
   		bfde4b54-0db7-4817-8032-87127bf19bb9 "Error en Impresion de datos en VarPR#" & Err.Number & " " & Err.Description
   		Err.Clear
   	End If
   	
   		If VarC(i) <> 0 Then
   	    	objExcel.Cells(i+4,6).Value = VarC(i)
   		End If
   		
   	If Err.Number <> 0 Then
   		bfde4b54-0db7-4817-8032-87127bf19bb9 "Error en Impresion de datos en VarC#" & Err.Number & " " & Err.Description
   		Err.Clear
   	End If
   	
   		If VarC(i) <> 0 And VarCLIStr(i) = " " Then
   	    	objExcel.Cells(i+4,6).Font.Bold = True
   		End If
   		
   	If Err.Number <> 0 Then
   		bfde4b54-0db7-4817-8032-87127bf19bb9 "Error en Impresion de datos en Bold2#" & Err.Number & " " & Err.Description
   		Err.Clear
   	End If
   	
   		If VarOPStr(i) <> " " Then
   	    	objExcel.Cells(i+4,7).Value = VarOPStr(i)
   	    	objExcel.Cells(i+4,8).Value = VarCicloOk(i)
   		End If
   		
   	If Err.Number <> 0 Then
   		bfde4b54-0db7-4817-8032-87127bf19bb9 "Error en Impresion de datos en OP#" & Err.Number & " " & Err.Description
   		Err.Clear
   	End If
   	
   	    If VarCicloOk(i) = "O" Then ' Rojo
   	    objExcel.Cells(i+4,9).Value = VarFallaStr(i)
   	    
   	    objExcel.Cells(i+4,7).Interior.Color = RGB(255, 125, 125)
   	    objExcel.Cells(i+4,6).Interior.Color = RGB(255, 125, 125)
   	    objExcel.Cells(i+4,5).Interior.Color = RGB(255, 125, 125)
   	    objExcel.Cells(i+4,4).Interior.Color = RGB(255, 125, 125)
   	    objExcel.Cells(i+4,3).Interior.Color = RGB(255, 125, 125)
   	    objExcel.Cells(i+4,2).Interior.Color = RGB(255, 125, 125)
   	    objExcel.Cells(i+4,1).Interior.Color = RGB(255, 125, 125)
   	    
   		End If
   		
   		If VarCicloOk(i) = "8" Then ' Rojo
   	    objExcel.Cells(i+4,9).Value = VarFallaStr(i)
   	    End If
   		
   		
   	If Err.Number <> 0 Then
   		bfde4b54-0db7-4817-8032-87127bf19bb9 "Error en Impresion de datos en VarFallaStr#" & Err.Number & " " & Err.Description
   		Err.Clear
   	End If
   	
   		If VarPR(i) = 12 Or VarPR(i) = 11  Or  VarCicloOk(i) = "8" Then ' Amarillo
   		    objExcel.Cells(i+4,7).Interior.Color = RGB(255, 238, 0)
   		    objExcel.Cells(i+4,6).Interior.Color = RGB(255, 238, 0)
   		    objExcel.Cells(i+4,5).Interior.Color = RGB(255, 238, 0)
   		    objExcel.Cells(i+4,4).Interior.Color = RGB(255, 238, 0)
   		    objExcel.Cells(i+4,3).Interior.Color = RGB(255, 238, 0)
   		    objExcel.Cells(i+4,2).Interior.Color = RGB(255, 238, 0)
   		    objExcel.Cells(i+4,1).Interior.Color = RGB(255, 238, 0)
   		End If
   		
   	End If
   Next
   
   	If Err.Number <> 0 Then
   		bfde4b54-0db7-4817-8032-87127bf19bb9 "Error en Impresion de datos en de lavados#" & Err.Number & " " & Err.Description
   		Err.Clear
   	End If
   
   ' Fin de impresion de datos en tabla
   
   objExcel.ActiveWorkbook.SaveAs NameInfDiario, 56
   objExcel.ActiveWorkbook.Close
   objExcel.Application.Quit
   
   
   Set objfso = CreateObject("Scripting.FileSystemObject")
   Do While objfso.FileExists(NameInfDiario) = False
   Loop
   k = Timer +5
   Do While (Timer<k)
   Loop	
   
   If Err.Number <> 0 Then
   	bfde4b54-0db7-4817-8032-87127bf19bb9 "Error en creacion de archivo excel#" & Err.Number & " " & Err.Description
   	Err.Clear
   End If
   
   bfde4b54-0db7-4817-8032-87127bf19bb9 "NameInfDiario#" & CStr(NameInfDiario)
   
   
   S23_Creador_InformeDiarioLavs_Gral = NameInfDiario

VB script "SA2_TotalTimeToString"
   Dim return, hora, minuto, segundo
   
   If Hour(thoras_) = 0 Then
   	hora = "00"
   Else
   	hora = CStr( dias_ * 24 + Hour(thoras_))
   End If
   
   If Minute(thoras_) = 0 Then
   	minuto = "00"
   Else
   	If Minute(thoras_) < 10 Then
   		minuto = "0" + CStr(Minute(thoras_))
   	Else
   		minuto = CStr(Minute(thoras_))
   	End If
   	
   End If
   
   If Second(thoras_) = 0 Then
   	segundo = "00"
   Else
   	If Second(thoras_) < 10 Then
   		segundo = "0" + CStr(Second(thoras_))
   	Else
   		segundo = CStr(Second(thoras_))
   	End If
   End If
   
   return = hora & ":" & minuto & ":" & segundo
   
   SA2_TotalTimeToString = return

VB script "S403_ActDia"
   	SmartTags("Ver_DIA_X") = Date()
   	SmartTags("Ver_DIA_XP") = Date()

VB script "S40_Write_Fall1BDD"
   If SmartTags("Lav1_grabFalla") Or SmartTags("Lav1_AlarmaVibracion") Then
   	
   Dim K
   
   'Declaration of local tags - Deklaration von lokalen Variablen
   Dim conn, rst, SQL_Table
   
   On Error Resume Next	
   	
   ' Recoleccion de datos de la lavadora 1 
   Dim hora, lav, falla
   
   'falla
   
   
   falla = SmartTags("Lav1_Falla")
   falla = S12_Conversor_BCD_to_Int(falla)
   If falla = 0 Then
   	K = Timer + 2
   	Do While (Timer<K)
   	Loop
   	
   End If
   
   falla = SmartTags("Lav1_Falla")
   falla = S12_Conversor_BCD_to_Int(falla)
   If falla = 0 Then
   	K = Timer + 2
   	Do While (Timer<K)
   	Loop
   	
   End If
   
   falla = SmartTags("Lav1_Falla")
   falla = S12_Conversor_BCD_to_Int(falla)
   
   If falla <> 0 Then
   	
   	hora = DateSerial(S12_Conversor_BCD_to_Int(SmartTags("Lav1_FchFll_Ano")), S12_Conversor_BCD_to_Int(SmartTags("Lav1_FchFll_Mes")), S12_Conversor_BCD_to_Int(SmartTags("Lav1_FchFll_Dia")))
   	hora = hora + TimeSerial(S12_Conversor_BCD_to_Int(SmartTags("Lav1_FchFll_Hr")), S12_Conversor_BCD_to_Int(SmartTags("Lav1_FchFll_Mins")), S12_Conversor_BCD_to_Int(SmartTags("Lav1_FchFll_segs")))
   	 
   		
   	'Lav
   	lav = 1
   	
   		Set conn = CreateObject("ADODB.Connection")
   	Set rst = CreateObject("ADODB.Recordset")
   	
   	'Abrir BBDD
   	conn.Open "Provider=MSDASQL;Initial Catalog=Lavadero;DSN=Lavadero"
   	
   	'Error routine
   	If Err.Number <> 0 Then
   		bfde4b54-0db7-4817-8032-87127bf19bb9 "S40_Lav1: Error abrirb base #" & Err.Number & " " & Err.Description
   		Err.Clear
   	End If
   	
   	'Definition of data record - Definition des Datensatzes
   	SQL_Table = "INSERT INTO FallasLavs VALUES ('"_
   		& hora 	& "' , '" _
   		& lav 	& "' , '" _
   		& falla	& "')"
   		
   	'Execute - Ausführen
   	Set rst = conn.Execute(SQL_Table)
   	
   	'Error routine - Fehler Routine
   	If Err.Number <> 0 Then
   		bfde4b54-0db7-4817-8032-87127bf19bb9 "S40_Error falla Lav1: #" & Err.Number & " " & Err.Description
   		Err.Clear
   		'Close data source - Datenquelle schließen
   		conn.close
   	End If
   	
   	Set rst = Nothing
   	Set conn = Nothing
   	
   	bfde4b54-0db7-4817-8032-87127bf19bb9 "Lav1: Falla grabada correctamente"
   	bfde4b54-0db7-4817-8032-87127bf19bb9 SQL_Table
   	'Tres confirmaciones diferentes si es que no se proceso la anterior, con loops se tilda
   
   	SmartTags("Lav1_ConfFalla") = True
   	K = Timer + 2
   	Do While (Timer<K)
   	Loop
   	If SmartTags("Lav1_Falla") <> 0 Then
   		SmartTags("Lav1_ConfFalla") = True
   	End If
   	
   	Else
   		bfde4b54-0db7-4817-8032-87127bf19bb9 "Lav1: Falla No grabada, No se leyo registro de falla del PLC"
   End If
   
   End If

VB script "S41_Write_Fall2BDD"
   If SmartTags("Lav2_grabFalla") Or SmartTags("Lav2_AlarmaVibracion") Then
   	
   Dim K
   
   'Declaration of local tags - Deklaration von lokalen Variablen
   Dim conn, rst, SQL_Table
   
   On Error Resume Next
   	
   ' Recoleccion de datos de la lavadora 1 
   Dim hora, lav, falla
   
   falla = SmartTags("Lav2_Falla")
   falla = S12_Conversor_BCD_to_Int(falla)
   If falla = 0 Then
   	K = Timer + 1
   	Do While (Timer<K)
   	Loop
   	
   End If
   
   falla = SmartTags("Lav2_Falla")
   falla = S12_Conversor_BCD_to_Int(falla)
   If falla = 0 Then
   	K = Timer + 1
   	Do While (Timer<K)
   	Loop
   	
   End If
   
   falla = SmartTags("Lav2_Falla")
   falla = S12_Conversor_BCD_to_Int(falla)
   
   If falla <> 0 Then
   '	
   	'hora actual
   	hora = DateSerial(S12_Conversor_BCD_to_Int(SmartTags("Lav2_FchFll_Ano")), S12_Conversor_BCD_to_Int(SmartTags("Lav2_FchFll_Mes")), S12_Conversor_BCD_to_Int(SmartTags("Lav2_FchFll_Dia")))
   	hora = hora + TimeSerial(S12_Conversor_BCD_to_Int(SmartTags("Lav2_FchFll_Hr")), S12_Conversor_BCD_to_Int(SmartTags("Lav2_FchFll_Mins")), S12_Conversor_BCD_to_Int(SmartTags("Lav2_FchFll_segs")))
   		
   	'Lav
   	lav = 2
   	
   	Set conn = CreateObject("ADODB.Connection")
   	Set rst = CreateObject("ADODB.Recordset")
   	
   	'Abrir BBDD
   	conn.Open "Provider=MSDASQL;Initial Catalog=Lavadero;DSN=Lavadero"
   	
   	'Error routine - Fehlerroutine
   	If Err.Number <> 0 Then
   		bfde4b54-0db7-4817-8032-87127bf19bb9 "S41_Lav2: Error abrirb base #" & Err.Number & " " & Err.Description
   		Err.Clear
   	End If
   		
   	
   	'Definition of data record - Definition des Datensatzes
   	SQL_Table = "INSERT INTO FallasLavs VALUES ('"_
   		& hora 	& "' , '" _
   		& lav 	& "' , '" _
   		& falla	& "')"
   	
   	'Execute - Ausführen
   	Set rst = conn.Execute(SQL_Table)
   	
   	'Error routine - Fehler Routine
   	If Err.Number <> 0 Then
   		bfde4b54-0db7-4817-8032-87127bf19bb9 "S41_Error falla Lav2: #" & Err.Number & " " & Err.Description
   		Err.Clear
   		'Close data source - Datenquelle schließen
   		conn.close
   	End If
   	
   		
   	Set rst = Nothing
   	Set conn = Nothing
   	
   		bfde4b54-0db7-4817-8032-87127bf19bb9 "Lav2: Falla grabada correctamente"
   		bfde4b54-0db7-4817-8032-87127bf19bb9 SQL_Table
   		'Tres confirmaciones diferentes si es que no se proceso la anterior, con loops se tilda
   	SmartTags("Lav2_ConfFalla") = True
   	K = Timer + 2
   	Do While (Timer<K)
   	Loop
   	If SmartTags("Lav2_Falla") <> 0 Then
   		SmartTags("Lav2_ConfFalla") = True
   	End If
   	
   	Else
   		bfde4b54-0db7-4817-8032-87127bf19bb9 "Lav2: Falla No grabada, No se leyo registro de falla del PLC"
   
   End If
   End If

VB script "S42_Write_Fall3BDD"
   If SmartTags("Lav3_grabFalla") Or SmartTags("Lav3_AlarmaVibracion") Then
   
   'Declaration of local tags - Deklaration von lokalen Variablen
   Dim conn, rst, SQL_Table, K
   
   On Error Resume Next
   
   ' Recoleccion de datos de la lavadora 1 
   Dim hora, lav, falla
   
   'falla
   falla =SmartTags("Lav3_Falla")
   falla = S12_Conversor_BCD_to_Int(falla)
   
   If falla = 0 Then
   	K = Timer + 1
   	Do While (Timer<K)
   	Loop
   	
   End If
   
   falla = SmartTags("Lav3_Falla")
   falla = S12_Conversor_BCD_to_Int(falla)
   If falla = 0 Then
   	K = Timer + 1
   	Do While (Timer<K)
   	Loop
   	
   End If
   falla = SmartTags("Lav3_Falla")
   falla = S12_Conversor_BCD_to_Int(falla)
   
   If falla <> 0 Then
   
   	Set conn = CreateObject("ADODB.Connection")
   	Set rst = CreateObject("ADODB.Recordset")
   	
   	'Abrir BBDD
   	conn.Open "Provider=MSDASQL;Initial Catalog=Lavadero;DSN=Lavadero"
   	
   	'Error routine - Fehlerroutine
   	If Err.Number <> 0 Then
   		bfde4b54-0db7-4817-8032-87127bf19bb9 "S42_Lav3: Error abrirb base #" & Err.Number & " " & Err.Description
   		Err.Clear
   	End If
   	
   	'hora actual
   	'hora = CStr(Date()) + " " + CStr(Time()) 
   		
   	hora = DateSerial(S12_Conversor_BCD_to_Int(SmartTags("Lav3_FchFll_Ano")), S12_Conversor_BCD_to_Int(SmartTags("Lav3_FchFll_Mes")), S12_Conversor_BCD_to_Int(SmartTags("Lav3_FchFll_Dia")))
   	hora = hora + TimeSerial(S12_Conversor_BCD_to_Int(SmartTags("Lav3_FchFll_Hr")), S12_Conversor_BCD_to_Int(SmartTags("Lav3_FchFll_Mins")), S12_Conversor_BCD_to_Int(SmartTags("Lav3_FchFll_segs")))
   	
   	'Lav
   	lav = 3
   	
   	
   	'Definition of data record - Definition des Datensatzes
   	SQL_Table = "INSERT INTO FallasLavs VALUES ('"_
   		& hora 	& "' , '" _
   		& lav 	& "' , '" _
   		& falla	& "')"
   		
   		'Execute - Ausführen
   	Set rst = conn.Execute(SQL_Table)
   	
   	'Error routine - Fehler Routine
   	If Err.Number <> 0 Then
   		bfde4b54-0db7-4817-8032-87127bf19bb9 "S42_Error falla Lav3: #" & Err.Number & " " & Err.Description
   		Err.Clear
   		'Close data source - Datenquelle schließen
   		conn.close
   	End If
   	
   		
   	Set rst = Nothing
   	Set conn = Nothing
   		bfde4b54-0db7-4817-8032-87127bf19bb9 "Lav3: Falla grabada correctamente"
   		bfde4b54-0db7-4817-8032-87127bf19bb9 SQL_Table
   		'Tres confirmaciones diferentes si es que no se proceso la anterior, con loops se tilda
   	SmartTags("Lav3_ConfFalla") = True
   	K = Timer + 2
   	Do While (Timer<K)
   	Loop
   	If SmartTags("Lav3_Falla") <> 0 Then
   		SmartTags("Lav3_ConfFalla") = True
   	End If
   	
   	Else
   		bfde4b54-0db7-4817-8032-87127bf19bb9 "Lav3: Falla No grabada, No se leyo registro de falla del PLC"
   
   End If
   End If

VB script "S18_Write_data_Lav4"
   Dim hayError, K
   hayError = False
   
   If SmartTags("Lav4_GrabarBDD") = True Then
   
   'Declaration of local tags - Deklaration von lokalen Variablen
   Dim conn, rst, SQL_Table
   
   On Error Resume Next
   
   Set conn = CreateObject("ADODB.Connection")
   Set rst = CreateObject("ADODB.Recordset")
   
   'Abrir BBDD
   conn.Open "Provider=MSDASQL;Initial Catalog=Lavadero;DSN=Lavadero"
   
   'Error routine
   If Err.Number <> 0 Then
   	bfde4b54-0db7-4817-8032-87127bf19bb9 "Lav4: Error abrirb base #" & Err.Number & " " & Err.Description
   	hayError = True
   End If
   	
   	
   ' Recoleccion de datos de la lavadora 4
   Dim fechafin, fechainicio, cliente_0, cliente_1, cliente_2, operario, carga, programa, ciclovalido, falla, valido_CN
   
   
   
   'fecha actual
   fechafin = DateSerial(S12_Conversor_BCD_to_Int(SmartTags("Lav4_FchFin_Ano")), S12_Conversor_BCD_to_Int(SmartTags("Lav4_FchFin_Mes")), S12_Conversor_BCD_to_Int(SmartTags("Lav4_FchFin_Dia")))
   fechafin = fechafin + TimeSerial(S12_Conversor_BCD_to_Int(SmartTags("Lav4_FchFin_Hr")), S12_Conversor_BCD_to_Int(SmartTags("Lav4_FchFin_Min")), S12_Conversor_BCD_to_Int(SmartTags("Lav4_FchFin_Seg")))
   
   'fecha de inicio del ciclo
   fechainicio = DateSerial(S12_Conversor_BCD_to_Int(SmartTags("Lav4_FchIni_Ano")), S12_Conversor_BCD_to_Int(SmartTags("Lav4_FchIni_Mes")), S12_Conversor_BCD_to_Int(SmartTags("Lav4_FchIni_Dia")))
   fechainicio = fechainicio + TimeSerial(S12_Conversor_BCD_to_Int(SmartTags("Lav4_FchIni_Hr")), S12_Conversor_BCD_to_Int(SmartTags("Lav4_FchIni_Min")), S12_Conversor_BCD_to_Int(SmartTags("Lav4_FchIni_Seg")))
   
   cliente_0 = SmartTags("Lav4_Cliente_0")
   cliente_1 = SmartTags("Lav4_Cliente_1")
   cliente_2 = SmartTags("Lav4_Cliente_2")
   	
   operario = SmartTags("Lav4_Operador")
   
   carga = SmartTags("Lav4_CantRopa")
   
   programa = S12_Conversor_BCD_to_Int(SmartTags("Lav4_Programa"))
   
   falla = SmartTags("Lav4_Falla")
   
   	If SmartTags("Lav4_St_Ciclo") = 0 Then
   		valido_CN = 1
   	Else
   		valido_CN = 0
   	End If
   
   	If SmartTags("Lav4_St_Ciclo") = 0 Or  S12_Conversor_BCD_to_Int(SmartTags("Lav4_St_Ciclo")) > 13 Then	
   		ciclovalido = 1
   	Else
   		ciclovalido = 0
   	End If
   
   'Definition of data record - Definition des Datensatzes
   SQL_Table = "INSERT INTO Lav4 VALUES ('"_
   	& fechafin 		& "' , '" _
   	& fechainicio 	& "' , '" _
   	& cliente_0 	& "' , '" _
   	& cliente_1 	& "' , '" _
   	& cliente_2 	& "' , '" _
   	& operario 		& "' , '" _
   	& carga 		& "' , '" _
   	& programa 		& "' , '" _
   	& ciclovalido & "' , '" _
   	& valido_CN & "')"
   
   If hayError = False Then
   	'Execute - Ausführen
   	Set rst = conn.Execute(SQL_Table)
   End If
   
   SmartTags("Lav4_Programa_Anterior") = SmartTags("Lav4_Programa")
   
   'Error routine - Fehler Routine
   If Err.Number <> 0 Then
   	bfde4b54-0db7-4817-8032-87127bf19bb9 "Error select Lav4: #" & Err.Number & " " & Err.Description
   	SmartTags("_errorNum4") = Err.Number
   	hayError = True
   End If
   
   If hayError = False Or SmartTags("Lav4_Cont_IntentosGrabado") >= 3 Then
   	'Tres confirmaciones diferentes si es que no se proceso la anterior, con loops se tilda
   	If SmartTags("Lav4_GrabarBDD") = True Then
   		SmartTags("Lav4_Ciclograbado") = True ' Quiere resetear una ves
   	End If
   	K = Timer + 2
   	Do While (Timer<K)
   	Loop
   	If SmartTags("Lav4_GrabarBDD") = True Then
   		SmartTags("Lav4_Ciclograbado") = True ' Quiere resetear dos veces
   	End If
   	K = Timer + 2
   	Do While (Timer<K)
   	Loop
   	If SmartTags("Lav4_GrabarBDD") = True Then ' Quiere resetear una tercera ves
   		SmartTags("Lav4_Ciclograbado") = True
   	End If
   	
   	If SmartTags("Lav4_Cont_IntentosGrabado") >= 3 Then
   		
   		'Envio email avisando que el ciclo no se grabo
   		cliente_0 = cliente_0 + "/" + cliente_1 + "/" + cliente_2
   		Call SA4_ErrorEnGrabBDD(4, fechafin, fechainicio, cliente_0,operario,carga,programa,ciclovalido)
   		
   		SmartTags("Lav4_Cont_IntentosGrabado") = 0
   		
   		If SmartTags("Lav4_GrabarBDD") = True Then
   			SmartTags("Lav4_Ciclograbado") = True ' Quiere resetear una cuarta ves
   		End If	
   	
   	End If
   
   		
   Else
   			
   		SmartTags("Lav4_Cont_IntentosGrabado") = SmartTags("Lav4_Cont_IntentosGrabado") + 1
   		
   End If
   
   
   End If
   	
   Err.Clear
   'Close data source
   Set conn = Nothing
   Set rst = Nothing 
   
   	
   
   	

VB script "S43_Write_Fall4BDD"
   If SmartTags("Lav4_grabFalla") Or SmartTags("Lav4_AlarmaVibracion") Then
   	
   	
   Dim hayError
   hayError = False
   
   Dim K
   
   'Declaration of local tags - Deklaration von lokalen Variablen
   Dim conn, rst, SQL_Table
   
   On Error Resume Next
   
   ' Recoleccion de datos de la lavadora 4 
   Dim hora, lav, falla
   
   'falla
   falla =SmartTags("Lav4_Falla")
   falla = S12_Conversor_BCD_to_Int(falla)
   
   If falla = 0 Then
   	K = Timer + 1
   	Do While (Timer<K)
   	Loop
   	
   End If
   
   falla = SmartTags("Lav4_Falla")
   falla = S12_Conversor_BCD_to_Int(falla)
   If falla = 0 Then
   	K = Timer + 1
   	Do While (Timer<K)
   	Loop
   	
   End If
   
   falla = SmartTags("Lav4_Falla")
   falla = S12_Conversor_BCD_to_Int(falla)
   	
   	If falla <> 0 Then
   	
   	Set conn = CreateObject("ADODB.Connection")
   	Set rst = CreateObject("ADODB.Recordset")
   	
   	'Abrir BBDD
   	conn.Open "Provider=MSDASQL;Initial Catalog=Lavadero;DSN=Lavadero"
   	
   	'Error routine - Fehlerroutine
   	If Err.Number <> 0 Then
   		bfde4b54-0db7-4817-8032-87127bf19bb9 "S43_Lav4: Error abrirb base #" & Err.Number & " " & Err.Description
   		Err.Clear
   	End If
   	
   	'hora actual
   	'hora = CStr(Date()) + " " + CStr(Time()) 
   	
   	hora = DateSerial(S12_Conversor_BCD_to_Int(SmartTags("Lav4_FchFll_Ano")), S12_Conversor_BCD_to_Int(SmartTags("Lav4_FchFll_Mes")), S12_Conversor_BCD_to_Int(SmartTags("Lav4_FchFll_Dia")))
   	hora = hora + TimeSerial(S12_Conversor_BCD_to_Int(SmartTags("Lav4_FchFll_Hr")), S12_Conversor_BCD_to_Int(SmartTags("Lav4_FchFll_Mins")), S12_Conversor_BCD_to_Int(SmartTags("Lav4_FchFll_segs")))
   	 
   	'Lav
   	lav = 4
   	
   	
   	'Definition of data record - Definition des Datensatzes
   	SQL_Table = "INSERT INTO FallasLavs VALUES ('"_
   		& hora 	& "' , '" _
   		& lav 	& "' , '" _
   		& falla	& "')"
   		
   	If hayError = False Then
   	'Execute - Ausführen
   		bfde4b54-0db7-4817-8032-87127bf19bb9 "S43_Error falla Lav4 grabada"
   		Set rst = conn.Execute(SQL_Table)
   	End If
   	'Error routine - Fehler Routine
   	If Err.Number <> 0 Then
   		bfde4b54-0db7-4817-8032-87127bf19bb9 "S43_Error falla Lav4: #" & Err.Number & " " & Err.Description
   		Err.Clear
   		'Close data source - Datenquelle schließen
   		conn.close
   	End If
   	
   	Set rst = Nothing
   	Set conn = Nothing
   		bfde4b54-0db7-4817-8032-87127bf19bb9 "Lav4: Falla grabada correctamente"
   		bfde4b54-0db7-4817-8032-87127bf19bb9 SQL_Table
   		'Tres confirmaciones diferentes si es que no se proceso la anterior, con loops se tilda
   	SmartTags("Lav4_ConfFalla") = True
   	K = Timer + 2
   	Do While (Timer<K)
   	Loop
   	If SmartTags("Lav4_Falla") <> 0 Then
   		SmartTags("Lav4_ConfFalla") = True
   	End If
   	
   	Else
   		bfde4b54-0db7-4817-8032-87127bf19bb9 "Lav4: Falla No grabada, No se leyo registro de falla del PLC"
   
   End If
   End If

VB script "S104_ActualizarCliEmPrincipal"
   'Declaracion de Variables locales
   Dim conn21, rst21, Consulta
   
   On Error Resume Next
   
   Set conn21 = CreateObject("ADODB.Connection")
   Set rst21 = CreateObject("ADODB.Recordset")
   
   'Abrir BDD
   conn21.Open "Provider=MSDASQL;Initial Catalog=Lavadero;DSN=Lavadero"
   
   
   'Chequeo de error
   If Err.Number <> 0 Then
   	bfde4b54-0db7-4817-8032-87127bf19bb9 "Error Conexion Actualización cliente en pantalla #" & Err.Number & " " & Err.Description
   	Err.Clear 
   	Set conn21 = Nothing
   	Exit Sub
   End If
   
   '	CONSULTA
   Consulta = "SELECT * FROM Cli_Lavadoras WHERE  ID = '" & SmartTags("Lav" & CStr(LavNro) & "_Cliente_" & CStr(CliNro)) &"';"
   'Ejecutar consulta
   Set rst21 = conn21.Execute(Consulta)
   SmartTags("Lav" & CStr(LavNro) & "_Cli_" & CStr(CliNro) & "_Str")= rst21.Fields(1).Value
   
   'Chequeo de error
   If Err.Number <> 0 Then
   	bfde4b54-0db7-4817-8032-87127bf19bb9 "Error Actualización cliente en pantalla #" & Err.Number & " " & Err.Description
   	Err.Clear 
   	Set conn21 = Nothing
   	Exit Sub
   End If
   	
   rst21.close
   conn21.close
   Set rst21 = Nothing
   Set conn21 = Nothing

VB script "SA3_Act_HoraFinEstPrincLav1"
   If SmartTags("Lav1_EnCiclo") = True Then
   	Dim fechainicio, K, tiempoDeCiclo
   	
   	K = Timer + 2
   	Do While (Timer<K)
   	Loop
   	
   	fechainicio = TimeSerial(S12_Conversor_BCD_to_Int(SmartTags("Lav1_FchIni_Hr")), S12_Conversor_BCD_to_Int(SmartTags("Lav1_FchIni_Min")), 00)
   	
   	Select Case S12_Conversor_BCD_to_Int(SmartTags("Lav1_Programa"))
   		Case 1
   			tiempoDeCiclo = 67
   		Case 2
   			tiempoDeCiclo = 71
   		Case 3
   			tiempoDeCiclo = 55
   		Case 4
   			tiempoDeCiclo = 75
   		Case 5
   			tiempoDeCiclo = 56
   		Case 6
   			tiempoDeCiclo = 88
   		Case 7
   			tiempoDeCiclo = 68
   		Case 8
   			tiempoDeCiclo = 74
   		Case 9
   			tiempoDeCiclo = 85
   		Case 10
   			tiempoDeCiclo = 61
   		Case 11
   			tiempoDeCiclo = 16
   		Case 12
   			tiempoDeCiclo = 16
   		Case 13
   			tiempoDeCiclo = 54
   		Case 14
   			tiempoDeCiclo = 68
   		Case 15
   			tiempoDeCiclo = 74
   		Case Else
   			tiempoDeCiclo = 00
   			
   	End Select
   
   	fechainicio = DateAdd("n",tiempoDeCiclo, fechainicio)
   	
   	SmartTags("Lav1_FinEstimado_Panel") = fechainicio
   	
   	If Err.Number <> 0 Then
   		bfde4b54-0db7-4817-8032-87127bf19bb9 "Error en Actualizacion de hora de fin panel#" & Err.Number & " " & Err.Description
   		Err.Clear
   	End If
   	
   	End If
   			

VB script "SA3_Act_HoraFinEstPrincLav2"
   If SmartTags("Lav2_EnCiclo") = True Then
   	Dim fechainicio, K, tiempoDeCiclo
   	
   	K = Timer + 2
   	Do While (Timer<K)
   	Loop
   	
   	fechainicio = TimeSerial(S12_Conversor_BCD_to_Int(SmartTags("Lav2_FchIni_Hr")), S12_Conversor_BCD_to_Int(SmartTags("Lav2_FchIni_Min")), 00)
   	
   	Select Case S12_Conversor_BCD_to_Int(SmartTags("Lav2_Programa"))
   		Case 1
   			tiempoDeCiclo = 67
   		Case 2
   			tiempoDeCiclo = 71
   		Case 3
   			tiempoDeCiclo = 55
   		Case 4
   			tiempoDeCiclo = 75
   		Case 5
   			tiempoDeCiclo = 56
   		Case 6
   			tiempoDeCiclo = 88
   		Case 7
   			tiempoDeCiclo = 68
   		Case 8
   			tiempoDeCiclo = 74
   		Case 9
   			tiempoDeCiclo = 85
   		Case 10
   			tiempoDeCiclo = 61
   		Case 11
   			tiempoDeCiclo = 16
   		Case 12
   			tiempoDeCiclo = 16
   		Case 13
   			tiempoDeCiclo = 54
   		Case 14
   			tiempoDeCiclo = 68
   		Case 15
   			tiempoDeCiclo = 74
   		Case Else
   			tiempoDeCiclo = 00
   			
   	End Select
   
   	fechainicio = DateAdd("n",tiempoDeCiclo, fechainicio)
   	
   	SmartTags("Lav2_FinEstimado_Panel") = fechainicio
   	
   	If Err.Number <> 0 Then
   		bfde4b54-0db7-4817-8032-87127bf19bb9 "Error en Actualizacion de hora de fin panel lav 2#" & Err.Number & " " & Err.Description
   		Err.Clear
   	End If
   	
   	End If
   			

VB script "SA3_Act_HoraFinEstPrincLav3"
   If SmartTags("Lav3_EnCiclo") = True Then
   	Dim fechainicio, K, tiempoDeCiclo
   	
   	K = Timer + 2
   	Do While (Timer<K)
   	Loop
   	
   	fechainicio = TimeSerial(S12_Conversor_BCD_to_Int(SmartTags("Lav3_FchIni_Hr")), S12_Conversor_BCD_to_Int(SmartTags("Lav3_FchIni_Min")), 00)
   	
   	Select Case S12_Conversor_BCD_to_Int(SmartTags("Lav3_Programa"))
   		Case 1
   			tiempoDeCiclo = 67
   		Case 2
   			tiempoDeCiclo = 71
   		Case 3
   			tiempoDeCiclo = 55
   		Case 4
   			tiempoDeCiclo = 75
   		Case 5
   			tiempoDeCiclo = 56
   		Case 6
   			tiempoDeCiclo = 88
   		Case 7
   			tiempoDeCiclo = 68
   		Case 8
   			tiempoDeCiclo = 74
   		Case 9
   			tiempoDeCiclo = 85
   		Case 10
   			tiempoDeCiclo = 61
   		Case 11
   			tiempoDeCiclo = 16
   		Case 12
   			tiempoDeCiclo = 16
   		Case 13
   			tiempoDeCiclo = 54
   		Case 14
   			tiempoDeCiclo = 68
   		Case 15
   			tiempoDeCiclo = 74
   		Case Else
   			tiempoDeCiclo = 00
   			
   	End Select
   
   	fechainicio = DateAdd("n",tiempoDeCiclo, fechainicio)
   	
   	SmartTags("Lav3_FinEstimado_Panel") = fechainicio
   	
   	If Err.Number <> 0 Then
   		bfde4b54-0db7-4817-8032-87127bf19bb9 "Error en Actualizacion de hora de fin panel Lav3#" & Err.Number & " " & Err.Description
   		Err.Clear
   	End If
   	
   End If
   			

VB script "SA3_Act_HoraFinEstPrincLav4"
   If SmartTags("Lav4_EnCiclo") = True Then
   	Dim fechainicio, K, tiempoDeCiclo
   	
   	K = Timer + 10
   	Do While (Timer<K)
   	Loop
   	
   	fechainicio = TimeSerial(S12_Conversor_BCD_to_Int(SmartTags("Lav4_FchIni_Hr")), S12_Conversor_BCD_to_Int(SmartTags("Lav4_FchIni_Min")), 00)
   	
   	Select Case S12_Conversor_BCD_to_Int(SmartTags("Lav4_Programa"))
   		Case 1
   			tiempoDeCiclo = 67
   		Case 2
   			tiempoDeCiclo = 71
   		Case 3
   			tiempoDeCiclo = 55
   		Case 4
   			tiempoDeCiclo = 75
   		Case 5
   			tiempoDeCiclo = 56
   		Case 6
   			tiempoDeCiclo = 88
   		Case 7
   			tiempoDeCiclo = 68
   		Case 8
   			tiempoDeCiclo = 74
   		Case 9
   			tiempoDeCiclo = 85
   		Case 10
   			tiempoDeCiclo = 61
   		Case 11
   			tiempoDeCiclo = 16
   		Case 12
   			tiempoDeCiclo = 16
   		Case 13
   			tiempoDeCiclo = 54
   		Case 14
   			tiempoDeCiclo = 68
   		Case 15
   			tiempoDeCiclo = 74
   		Case Else
   			tiempoDeCiclo = 00
   			
   	End Select
   
   	fechainicio = DateAdd("n",tiempoDeCiclo, fechainicio)
   	
   	SmartTags("Lav4_FinEstimado_Panel") = fechainicio
   	
   	If Err.Number <> 0 Then
   		bfde4b54-0db7-4817-8032-87127bf19bb9 "Error en Actualizacion de hora de fin panel Lav4#" & Err.Number & " " & Err.Description
   		Err.Clear
   	End If
   			
   End If
   			

VB script "S400_ActListLav"
   bfde4b54-0db7-4817-8032-87127bf19bb9 "Entro a S400"
   'Declaracion de Variables locales
   Dim connListLav, rstListLav, SQL_Table
   Dim Consulta, Dia, i
   
   Dim cantDeRegistros
   cantDeRegistros = 20
   
   Dim cli0(20), cli1(20), cli2(20), ope(20), band_1(20), VarCliStr(20), VarOPStr(20)
   
   For i = 1 To cantDeRegistros
   	SmartTags("Ver_Cli_Str_" & CStr(i - 1))			= "-"
   	SmartTags("Ver_Operador_Str_" & CStr(i - 1))	= "-"
   Next
   
   On Error Resume Next
   
   Set connListLav = CreateObject("ADODB.Connection")
   'Abrir BDD
   connListLav.Open "Provider=MSDASQL;Initial Catalog=Lavadero;DSN=Lavadero"
   
   bfde4b54-0db7-4817-8032-87127bf19bb9 "Entro a S400_1"
   'Chequeo de error
   If Err.Number <> 0 Then
   	bfde4b54-0db7-4817-8032-87127bf19bb9 "Error al abrir BDD#" & Err.Number & " " & Err.Description
   	Err.Clear 
   	connListLav.close
   	Exit Sub
   End If
   
   If (SmartTags("Ver_IDList") < 0) Then
   	SmartTags("Ver_IDList") = 0
   End If
   
   bfde4b54-0db7-4817-8032-87127bf19bb9 "Entro a S400_2"
   'Chequeo de error
   If Err.Number <> 0 Then
   	bfde4b54-0db7-4817-8032-87127bf19bb9 "Error al abrir BDD#" & Err.Number & " " & Err.Description
   	Err.Clear 
   	connListLav.close
   	Exit Sub
   	
   End If
   
   Dia = SmartTags("Ver_DIA_X")
   
   	Consulta = "SELECT * FROM Lav" & CStr(LavNro) & " WHERE cast(fechafin As Date) = '"
   	Consulta = Consulta & CStr(Year(Dia)) & "-" & CStr(Month(Dia)) & "-" & CStr(Day(Dia)) & "' "
   	Consulta = Consulta & "order by fechafin"
   	
   	bfde4b54-0db7-4817-8032-87127bf19bb9 "Entro a S400_3"
   Set rstListLav = CreateObject("ADODB.Recordset")
   'Ejecutar consulta
   Set rstListLav = connListLav.Execute(Consulta)
   
   'Salteo registros segun indice
   If SmartTags("Ver_IDList") <> 0 Then
   	For i = 1 To SmartTags("Ver_IDList")
   		rstListLav.MoveNext
   	Next
   End If
   
   bfde4b54-0db7-4817-8032-87127bf19bb9 "Entro a S400_4"
   
   
   'Llenado de variables que muestan la lista
   For i = 1 To cantDeRegistros
   	
   	If rstListLav.EOF = False Then
   		SmartTags("Ver_HoraFin_" & CStr(i - 1)) 	= rstListLav.Fields(0).Value
   		SmartTags("Ver_HoraInicio_" & CStr(i - 1)) 	= rstListLav.Fields(1).Value
   		cli0(i)										= rstListLav.Fields(2).Value
   		cli1(i)										= rstListLav.Fields(3).Value
   		cli2(i)										= rstListLav.Fields(4).Value
   		ope(i)										= rstListLav.Fields(5).Value
   		SmartTags("Ver_Carga_" & CStr(i - 1)) 		= rstListLav.Fields(6).Value
   		SmartTags("Ver_Programa_" & CStr(i - 1))	= rstListLav.Fields(7).Value
   		SmartTags("Ver_CicloValido_" & CStr(i - 1))	= rstListLav.Fields(8).Value
   		
   		rstListLav.MoveNext
   	Else	
   		SmartTags("Ver_HoraFin_" & CStr(i - 1)) 	= 0
   		SmartTags("Ver_HoraInicio_" & CStr(i - 1)) 	= 0
   		cli0(i)										= 0
   		cli1(i)										= 0
   		cli2(i)										= 0
   		ope(i)										= 0
   		SmartTags("Ver_Carga_" & CStr(i - 1)) 		= 0
   		SmartTags("Ver_Programa_" & CStr(i - 1))	= 0
   		SmartTags("Ver_CicloValido_" & CStr(i - 1))	= False
   	End If
   Next
   
   If Err.Number <> 0 Then
   	bfde4b54-0db7-4817-8032-87127bf19bb9 "Error en grabar los datos en variables" & Err.Number & " " & Err.Description
   	Err.Clear
   
   	rstListLav.close
   	connListLav.close 
   	Exit Sub
   End If
   
   bfde4b54-0db7-4817-8032-87127bf19bb9 "Entro a S400_5"
   ' ######### Consulta para obtener el listado actualizado de clientes ############
   
   Dim rstcli, rstope, ConsultaCli, ConsultaOpe, j
   
   ConsultaCli = "SELECT * FROM Cli_Lavadoras;"
   
   Set rstcli = CreateObject("ADODB.Recordset")
   'Ejecutar consulta
   Set rstcli = connListLav.Execute(ConsultaCli)
   ''''''''''''''''''''''''''''''''''''''''''''''''''''''''''''''''''''''''''''''''
   
   ' ######### Consulta para obtener el listado actualizado de OPERADORES ############
   
   ConsultaOpe = "SELECT * FROM Op_Lavadoras;"
   
   Set rstope = CreateObject("ADODB.Recordset")
   'Ejecutar consulta
   Set rstope = connListLav.Execute(ConsultaOpe)
   ''''''''''''''''''''''''''''''''''''''''''''''''''''''''''''''''''''''''''''''''
   
   ' Establecer los clientes
   For i = 1 To cantDeRegistros
   	band_1(i)		= 0
   Next
   bfde4b54-0db7-4817-8032-87127bf19bb9 "Entro a S400_6"
   Do While rstcli.EOF = False
   	For j = 1 To cantDeRegistros 
   		If (rstcli.Fields(0).Value = cli0(j)) Then 
   			If band_1(j) = 0 Then
   				VarCliStr(j) = Trim(rstcli.Fields(1).Value)
   				band_1(j) = 1
   			Else
   				VarCliStr(j) = VarCliStr(j) + "/" + Trim(rstcli.Fields(1).Value)
   			End If
   		End If
   
   		If (rstcli.Fields(0).Value = cli1(j)) Then
   			If band_1(j) = 0 Then
   				VarCliStr(j) = Trim(rstcli.Fields(1).Value)
   				band_1(j) = 1
   			Else
   				VarCliStr(j) = VarCliStr(j) + "/" + Trim(rstcli.Fields(1).Value)
   			End If
   		End If
   
   		If (rstcli.Fields(0).Value = cli2(j)) Then
   			If band_1(j) = 0 Then
   				VarCliStr(j) = Trim(rstcli.Fields(1).Value)
   				band_1(j) = 1
   			Else
   				VarCliStr(j) = VarCliStr(j) + "/" + Trim(rstcli.Fields(1).Value)
   			End If
   		End If
   		
   	Next
   	rstcli.MoveNext
   Loop
   bfde4b54-0db7-4817-8032-87127bf19bb9 "Entro a S400_7"
   
   If Err.Number <> 0 Then
   	bfde4b54-0db7-4817-8032-87127bf19bb9 "Error en establecer los clientes#" & Err.Number & " " & Err.Description
   	Err.Clear
   	rstcli.close
   	rstope.close
   	rstListLav.close
   	connListLav.close 
   	Exit Sub
   End If
   
   ' Establecer los operarios
   Do While rstope.EOF = False
   	For j = 1 To cantDeRegistros
   		If (rstope.Fields(0).Value = ope(j)) Then
   			VarOPStr(j) = Trim(rstope.Fields(1).Value)
   		End If
   	Next
   	rstope.MoveNext
   Loop
   bfde4b54-0db7-4817-8032-87127bf19bb9 "Entro a S400_8"
   If Err.Number <> 0 Then
   	bfde4b54-0db7-4817-8032-87127bf19bb9 "Error en establecer los operadores#" & Err.Number & " " & Err.Description
   	Err.Clear
   	rstcli.close
   	rstope.close
   	rstListLav.close
   	connListLav.close
   	Exit Sub
   End If
   
   For i = 1 To cantDeRegistros
   		SmartTags("Ver_Cli_Str_" & CStr(i - 1))			=  CStr(VarCliStr(i))
   		SmartTags("Ver_Operador_Str_" & CStr(i - 1))	= CStr(VarOPStr (i))
   Next
   
   bfde4b54-0db7-4817-8032-87127bf19bb9 "Entro a S400_9"
   '########################################################################
   rstcli.close
   rstope.close
   rstListLav.close
   connListLav.close
   
   Set rstcli = Nothing
   Set rstope = Nothing
   Set rstListLav = Nothing
   Set connListLav = Nothing
   
   If Err.Number <> 0 Then
   	bfde4b54-0db7-4817-8032-87127bf19bb9 "Error en establecer los operadores#" & Err.Number & " " & Err.Description
   	Err.Clear
   	rstcli.close
   	rstope.close
   	rstListLav.close
   	connListLav.close
   	Exit Sub
   End If
   
   bfde4b54-0db7-4817-8032-87127bf19bb9 "Salio a S400"

VB script "S03_Write_data_record_into_a_table"
   '////////////////////////////////////////////////////////////////
   ' en: The script wirtes the indicated data record into a table
   ' de: Das Skript schreibt den angegebene Datensatz in eine Tabelle
   ' Created: 19-07-2012
   ' Version: v1.0
   ' Author:  HH 
   '////////////////////////////////////////////////////////////////
   
   'Declaration of local tags - Deklaration von lokalen Variablen
   Dim conn, rst, SQL_Table, berni, fechapl, fecha, hora
   
   On Error Resume Next
   
   If SmartTags("Cada15M") Then 
   Set conn = CreateObject("ADODB.Connection")
   Set rst = CreateObject("ADODB.Recordset")
   
   'Open data source - Datenquelle öffnen
   conn.Open "Provider=MSDASQL;Initial Catalog=Lavadero;DSN=Lavadero"
   'conn.Open "Provider=MSDASQL;Initial Catalog=" & SmartTags("szDatabase") & ";DSN="&Database_Name&"" 'DSN= name of the odbc database - DSN= Name der ODBC-Datenbank
   
   'Error routine - Fehlerroutine
   If Err.Number <> 0 Then
   	bfde4b54-0db7-4817-8032-87127bf19bb9 "Error abrirb base #" & Err.Number & " " & Err.Description
   	Err.Clear
   	Set conn = Nothing 
   	Exit Sub
   End If
   
   
   
   	'Definition of data record - Definition des Datensatzes
   	SQL_Table = "INSERT INTO Plancha1 VALUES ('"_
   		& SmartTags("Planchadora1_FechaHoraPLC")_
   		& "' , '" & SmartTags("Planchadora1_TiempoTotal")_
   		& "' , '" & SmartTags("Planchadora1_ProductividadTotal")_
   	  	& "' , '" & SmartTags("Planchadora1_RendimientoTotal")_
   	  	& "' , '" & SmartTags("Planchadora1_RendPesado")_	 
   	  	& "' , '" & SmartTags("Planchadora1_Supervisores{1}_Tiempo")_
   	  	& "' , '" & SmartTags("Planchadora1_Supervisores{1}_Produccion")_
   	  	& "' , '" & SmartTags("Planchadora1_Supervisores{1}_Rendimiento")_
   	  	& "' , '" & SmartTags("Planchadora1_Supervisores{1}_RendPesado")_
   	  	& "' , '" & SmartTags("Planchadora1_Supervisores{2}_Tiempo")_
   	  	& "' , '" & SmartTags("Planchadora1_Supervisores{2}_Produccion")_
   	  	& "' , '" & SmartTags("Planchadora1_Supervisores{2}_Rendimiento")_
   	  	& "' , '" & SmartTags("Planchadora1_Supervisores{2}_RendPesado")_
   		& "' , '" & SmartTags("Planchadora1_Supervisores{3}_Tiempo")_
   		& "' , '" & SmartTags("Planchadora1_Supervisores{3}_Produccion")_
   		& "' , '" & SmartTags("Planchadora1_Supervisores{3}_Rendimiento")_
   		& "' , '" & SmartTags("Planchadora1_Supervisores{3}_RendPesado")_
   		& "' , '" & SmartTags("Planchadora1_Supervisores{4}_Tiempo")_
   		& "' , '" & SmartTags("Planchadora1_Supervisores{4}_Produccion")_
   		& "' , '" & SmartTags("Planchadora1_Supervisores{4}_Rendimiento")_
   		& "' , '" & SmartTags("Planchadora1_Supervisores{4}_RendPesado")_
   		& "' , '" & SmartTags("Planchadora1_Operadores{1}_Tiempo")_
   		& "' , '" & SmartTags("Planchadora1_Operadores{1}_Produccion")_
   		& "' , '" & SmartTags("Planchadora1_Operadores{1}_Rendimiento")_
   		& "' , '" & SmartTags("Planchadora1_Operadores{1}_RendPesado")_	  
   		& "' , '" & SmartTags("Planchadora1_Operadores{2}_Tiempo")_
   		& "' , '" & SmartTags("Planchadora1_Operadores{2}_Produccion")_
   		& "' , '" & SmartTags("Planchadora1_Operadores{2}_Rendimiento")_
   		& "' , '" & SmartTags("Planchadora1_Operadores{2}_RendPesado")_		  
   		& "' , '" & SmartTags("Planchadora1_Operadores{3}_Tiempo")_
   		& "' , '" & SmartTags("Planchadora1_Operadores{3}_Produccion")_
   		& "' , '" & SmartTags("Planchadora1_Operadores{3}_Rendimiento")_
   		& "' , '" & SmartTags("Planchadora1_Operadores{3}_RendPesado")_	
   		& "' , '" & SmartTags("Planchadora1_Operadores{4}_Tiempo")_
   		& "' , '" & SmartTags("Planchadora1_Operadores{4}_Produccion")_
   		& "' , '" & SmartTags("Planchadora1_Operadores{4}_Rendimiento")_
   		& "' , '" & SmartTags("Planchadora1_Operadores{4}_RendPesado")_	
   		& "' , '" & SmartTags("Planchadora1_Operadores{5}_Tiempo")_
   		& "' , '" & SmartTags("Planchadora1_Operadores{5}_Produccion")_
   		& "' , '" & SmartTags("Planchadora1_Operadores{5}_Rendimiento")_
   		& "' , '" & SmartTags("Planchadora1_Operadores{5}_RendPesado")_	
   		& "' , '" & SmartTags("Planchadora1_Operadores{6}_Tiempo")_
   		& "' , '" & SmartTags("Planchadora1_Operadores{6}_Produccion")_
   		& "' , '" & SmartTags("Planchadora1_Operadores{6}_Rendimiento")_
   		& "' , '" & SmartTags("Planchadora1_Operadores{6}_RendPesado")_	
   		& "' , '" & SmartTags("Planchadora1_Operadores{7}_Tiempo")_
   		& "' , '" & SmartTags("Planchadora1_Operadores{7}_Produccion")_
   		& "' , '" & SmartTags("Planchadora1_Operadores{7}_Rendimiento")_
   		& "' , '" & SmartTags("Planchadora1_Operadores{7}_RendPesado")_	
   		& "' , '" & SmartTags("Planchadora1_Operadores{8}_Tiempo")_
   		& "' , '" & SmartTags("Planchadora1_Operadores{8}_Produccion")_
   		& "' , '" & SmartTags("Planchadora1_Operadores{8}_Rendimiento")_
   		& "' , '" & SmartTags("Planchadora1_Operadores{8}_RendPesado")_	
   		& "' , '" & SmartTags("Planchadora1_Operadores{9}_Tiempo")_
   		& "' , '" & SmartTags("Planchadora1_Operadores{9}_Produccion")_
   		& "' , '" & SmartTags("Planchadora1_Operadores{9}_Rendimiento")_
   		& "' , '" & SmartTags("Planchadora1_Operadores{9}_RendPesado")_	
   		& "' , '" & SmartTags("Planchadora1_Operadores{10}_Tiempo")_
   		& "' , '" & SmartTags("Planchadora1_Operadores{10}_Produccion")_
   		& "' , '" & SmartTags("Planchadora1_Operadores{10}_Rendimiento")_
   		& "' , '" & SmartTags("Planchadora1_Operadores{10}_RendPesado")_	
   		& "' , '" & SmartTags("Planchadora1_Supervisores{1}_Estado")_
   		& "' , '" & SmartTags("Planchadora1_Supervisores{2}_Estado")_
   		& "' , '" & SmartTags("Planchadora1_Supervisores{3}_Estado")_
   		& "' , '" & SmartTags("Planchadora1_Supervisores{4}_Estado")_
   		& "' , '" & SmartTags("Planchadora1_Operadores{1}_Estado")_
   		& "' , '" & SmartTags("Planchadora1_Operadores{2}_Estado")_
   		& "' , '" & SmartTags("Planchadora1_Operadores{3}_Estado")_
   		& "' , '" & SmartTags("Planchadora1_Operadores{4}_Estado")_
   		& "' , '" & SmartTags("Planchadora1_Operadores{5}_Estado")_
   		& "' , '" & SmartTags("Planchadora1_Operadores{6}_Estado")_
   		& "' , '" & SmartTags("Planchadora1_Operadores{7}_Estado")_
   		& "' , '" & SmartTags("Planchadora1_Operadores{8}_Estado")_
   		& "' , '" & SmartTags("Planchadora1_Operadores{9}_Estado")_
   		& "' , '" & SmartTags("Planchadora1_Operadores{10}_Estado")_
   		& "' , '" & SmartTags("Planchadora1_SumaOperario")_
   		& "' , '" & SmartTags("Planchadora1_WeekDay")_
   		& "')"
   	' & _"' , '" & SmartTags("nValue_1") & "' , '" & SmartTags("nValue_2") & _"' , '" & SmartTags("nValue_3") & "')"
   	'Insert the data reacord of the table - Datensatz in die Tabelle hinzufügen
   '	Set rst = conn.Execute(SQL_Table)
   	
   'SQL_Table = "SELECT * FROM Plancha2 WHERE Nr = " & SmartTags("nDat_No")  '* = Alle Daten '* = all data
   
   'Execute - Ausführen
   Set rst = conn.Execute(SQL_Table)
   
   'Error routine - Fehler Routine
   If Err.Number <> 0 Then
   	bfde4b54-0db7-4817-8032-87127bf19bb9 "Error select Plancha1 #" & Err.Number & " " & Err.Description
   	Err.Clear
   	'Close data source - Datenquelle schließen
   	conn.close
       Set conn = Nothing
   	Set rst = Nothing 
   	Exit Sub
   End If
   	
   	'Definition of data record - Definition des Datensatzes
   	
   SQL_Table = "INSERT INTO Plancha2 VALUES ('"_
   		& SmartTags("Planchadora1_FechaHoraPLC")_
   		& "' , '" & SmartTags("Planchadora2_TiempoTotal")_
   		& "' , '" & SmartTags("Planchadora2_ProductividadTotal")_
   		& "' , '" & SmartTags("Planchadora2_RendimientoTotal")_
   		& "' , '" & SmartTags("Planchadora2_RendPesado")_  
   		& "' , '" & SmartTags("Planchadora2_Supervisores{1}_Tiempo")_
   		& "' , '" & SmartTags("Planchadora2_Supervisores{1}_Produccion")_
   		& "' , '" & SmartTags("Planchadora2_Supervisores{1}_Rendimiento")_
   		& "' , '" & SmartTags("Planchadora2_Supervisores{1}_RendPesado")_	  
   		& "' , '" & SmartTags("Planchadora2_Supervisores{2}_Tiempo")_
   		& "' , '" & SmartTags("Planchadora2_Supervisores{2}_Produccion")_
   		& "' , '" & SmartTags("Planchadora2_Supervisores{2}_Rendimiento")_
   		& "' , '" & SmartTags("Planchadora2_Supervisores{2}_RendPesado")_		  
   		& "' , '" & SmartTags("Planchadora2_Supervisores{3}_Tiempo")_
   		& "' , '" & SmartTags("Planchadora2_Supervisores{3}_Produccion")_
   		& "' , '" & SmartTags("Planchadora2_Supervisores{3}_Rendimiento")_
   		& "' , '" & SmartTags("Planchadora2_Supervisores{3}_RendPesado")_	
   		& "' , '" & SmartTags("Planchadora2_Supervisores{4}_Tiempo")_
   		& "' , '" & SmartTags("Planchadora2_Supervisores{4}_Produccion")_
   		& "' , '" & SmartTags("Planchadora2_Supervisores{4}_Rendimiento")_
   		& "' , '" & SmartTags("Planchadora2_Supervisores{4}_RendPesado")_	
   		& "' , '" & SmartTags("Planchadora2_Operadores{1}_Tiempo")_
   		& "' , '" & SmartTags("Planchadora2_Operadores{1}_Produccion")_
   		& "' , '" & SmartTags("Planchadora2_Operadores{1}_Rendimiento")_
   		& "' , '" & SmartTags("Planchadora2_Operadores{1}_RendPesado")_	  
   		& "' , '" & SmartTags("Planchadora2_Operadores{2}_Tiempo")_
   		& "' , '" & SmartTags("Planchadora2_Operadores{2}_Produccion")_
   		& "' , '" & SmartTags("Planchadora2_Operadores{2}_Rendimiento")_
   		& "' , '" & SmartTags("Planchadora2_Operadores{2}_RendPesado")_
   		& "' , '" & SmartTags("Planchadora2_Operadores{3}_Tiempo")_
   		& "' , '" & SmartTags("Planchadora2_Operadores{3}_Produccion")_
   		& "' , '" & SmartTags("Planchadora2_Operadores{3}_Rendimiento")_
   		& "' , '" & SmartTags("Planchadora2_Operadores{3}_RendPesado")_
   		& "' , '" & SmartTags("Planchadora2_Operadores{4}_Tiempo")_
   		& "' , '" & SmartTags("Planchadora2_Operadores{4}_Produccion")_
   		& "' , '" & SmartTags("Planchadora2_Operadores{4}_Rendimiento")_
   		& "' , '" & SmartTags("Planchadora2_Operadores{4}_RendPesado")_
   		& "' , '" & SmartTags("Planchadora2_Operadores{5}_Tiempo")_
   		& "' , '" & SmartTags("Planchadora2_Operadores{5}_Produccion")_
   		& "' , '" & SmartTags("Planchadora2_Operadores{5}_Rendimiento")_
   		& "' , '" & SmartTags("Planchadora2_Operadores{5}_RendPesado")_
   		& "' , '" & SmartTags("Planchadora2_Operadores{6}_Tiempo")_
   		& "' , '" & SmartTags("Planchadora2_Operadores{6}_Produccion")_
   		& "' , '" & SmartTags("Planchadora2_Operadores{6}_Rendimiento")_
   		& "' , '" & SmartTags("Planchadora2_Operadores{6}_RendPesado")_
   		& "' , '" & SmartTags("Planchadora2_Operadores{7}_Tiempo")_
   		& "' , '" & SmartTags("Planchadora2_Operadores{7}_Produccion")_
   		& "' , '" & SmartTags("Planchadora2_Operadores{7}_Rendimiento")_
   		& "' , '" & SmartTags("Planchadora2_Operadores{7}_RendPesado")_
   		& "' , '" & SmartTags("Planchadora2_Operadores{8}_Tiempo")_
   		& "' , '" & SmartTags("Planchadora2_Operadores{8}_Produccion")_
   		& "' , '" & SmartTags("Planchadora2_Operadores{8}_Rendimiento")_
   		& "' , '" & SmartTags("Planchadora2_Operadores{8}_RendPesado")_
   		& "' , '" & SmartTags("Planchadora2_Operadores{9}_Tiempo")_
   		& "' , '" & SmartTags("Planchadora2_Operadores{9}_Produccion")_
   		& "' , '" & SmartTags("Planchadora2_Operadores{9}_Rendimiento")_
   		& "' , '" & SmartTags("Planchadora2_Operadores{9}_RendPesado")_
   		& "' , '" & SmartTags("Planchadora2_Operadores{10}_Tiempo")_
   		& "' , '" & SmartTags("Planchadora2_Operadores{10}_Produccion")_
   		& "' , '" & SmartTags("Planchadora2_Operadores{10}_Rendimiento")_
   		& "' , '" & SmartTags("Planchadora2_Operadores{10}_RendPesado")_
   		& "' , '" & SmartTags("Planchadora2_Supervisores{1}_Estado")_
   		& "' , '" & SmartTags("Planchadora2_Supervisores{2}_Estado")_
   		& "' , '" & SmartTags("Planchadora2_Supervisores{3}_Estado")_
   		& "' , '" & SmartTags("Planchadora2_Supervisores{4}_Estado")_
   		& "' , '" & SmartTags("Planchadora2_Operadores{1}_Estado")_
   		& "' , '" & SmartTags("Planchadora2_Operadores{2}_Estado")_
   		& "' , '" & SmartTags("Planchadora2_Operadores{3}_Estado")_
   		& "' , '" & SmartTags("Planchadora2_Operadores{4}_Estado")_
   		& "' , '" & SmartTags("Planchadora2_Operadores{5}_Estado")_
   		& "' , '" & SmartTags("Planchadora2_Operadores{6}_Estado")_
   		& "' , '" & SmartTags("Planchadora2_Operadores{7}_Estado")_
   		& "' , '" & SmartTags("Planchadora2_Operadores{8}_Estado")_
   		& "' , '" & SmartTags("Planchadora2_Operadores{9}_Estado")_
   		& "' , '" & SmartTags("Planchadora2_Operadores{10}_Estado")_
   		& "' , '" & SmartTags("Planchadora2_SumaOperario")_
   		& "' , '" & SmartTags("Planchadora2_WeekDay")_
   		& "')"
    
    	' & _"' , '" & SmartTags("nValue_1") & "' , '" & SmartTags("nValue_2") & _"' , '" & SmartTags("nValue_3") & "')"
   	'Insert the data reacord of the table - Datensatz in die Tabelle hinzufügen
   Set rst = conn.Execute(SQL_Table)
   
   
   'Error routine - Fehler Routine
   If Err.Number <> 0 Then
   	bfde4b54-0db7-4817-8032-87127bf19bb9 "Error select Plancha2 #" & Err.Number & " " & Err.Description
   	Err.Clear
   	'Close data source - Datenquelle schließen
   	conn.close
       Set conn = Nothing
   	Set rst = Nothing 
   	Exit Sub
   End If
   	
   
   'Close data source - Datenquelle schließen
   conn.close
   
   Set rst = Nothing
   Set conn = Nothing
   
   End If

VB script "SA4_ErrorEnGrabBDD"
   Dim appOutlook 'As OUTLOOK.APPLICATION
   Dim mlNewMail 'As MailItem
   Dim objEntry
   Dim Text, valido_str
   	
   Const addressee = "crj@eprocsrl.com.ar; danielst@live.com.ar;"' josemariacullen@hotmail.com; zekeserio@hotmail.com;"	
   
   '## ENVIAR Aviso POR EMAIL AVISO NO SE PUDO GRABAR CICLO
   
   If valido = 1 Then
   	valido_str = "Sî"
   Else
   	valido_str = "No"
   End If
   
   		
   	' Text to be sent 
   	
   	Text = "AVISO DE FALLA DE GRABADO DE CICLO EN LAVADORA " + CStr(LavNro) + vbCrLf +_
   			"Hora Fin: " + CStr(Date()) + " " + CStr(fechafin) + vbCrLf +_
   			"Hora Inicio: " + CStr(fechainicio) + vbCrLf +_
   			"Clientes: " + CStr(cli) + vbCrLf +_
   			"Operario: " + CStr(operario) + vbCrLf +_
   			"Carga: " + CStr(carga/10) + " Kg" + vbCrLf +_
   			"Programa: " + CStr(programa) + vbCrLf +_
   			"Valido: " + valido_str + vbCrLf +_
   			"Error: #" & SmartTags("_errorNum" & CStr(LavNro))
   			
   			Err.Clear
   	
   	Set appOutlook = CreateObject("OUTLOOK.APPLICATION")
   	
   	
   	'Generating and sending an e-mail:
   	Set mlNewMail = appOutlook.CreateItem(0)
   	mlNewMail.Display
   	mlNewMail.To = addressee
   	mlNewMail.Subject = "Aviso de error en grabado de base de datos en Lav Nro " + CStr(LavNro)
   	mlNewMail.Body = Text
   	mlNewMail.save
   	mlNewMail.send 
   	

VB script "S401_EditarLavado"
   bfde4b54-0db7-4817-8032-87127bf19bb9 "Entro a S402"
   
   'Declaracion de variables locales
   Dim conn302, rst302, SQL_Table
   Dim Dia, fechafin, fechainicio, cli1, cli2, cli3, ope, carga, programa, ciclovalido
   Dim fechafin_ans
   
   On Error Resume Next
   
   Set conn302 = CreateObject("ADODB.Connection")
   Set rst302 = CreateObject("ADODB.Recordset")
   
   'Abrir BBDD
   conn302.Open "Provider=MSDASQL;Initial Catalog=Lavadero;DSN=Lavadero"
   
   Dia = SmartTags("Ver_DIA_X")
   
   fechafin_ans = DateSerial(Year(Dia), Month(Dia), Day(Dia)) + TimeSerial(Hour(SmartTags("Ver_HoraFin_X_ans")), Minute(SmartTags("Ver_HoraFin_X_ans")), Second(SmartTags("Ver_HoraFin_X_ans")))
   
   'Nuevos Registros
   fechafin 	= DateSerial(Year(Dia), Month(Dia), Day(Dia)) + TimeSerial(Hour(SmartTags("Ver_HoraFin_X")), Minute(SmartTags("Ver_HoraFin_X")), Second(SmartTags("Ver_HoraFin_X")))
   fechainicio = DateSerial(Year(Dia), Month(Dia), Day(Dia)) + TimeSerial(Hour(SmartTags("Ver_HoraInicio_X")), Minute(SmartTags("Ver_HoraInicio_X")), Second(SmartTags("Ver_HoraInicio_X")))
   cli1 		= SmartTags("Ver_Cli1_Str_X")
   cli2 		= SmartTags("Ver_Cli2_Str_X")
   cli3 		= SmartTags("Ver_Cli3_Str_X")
   ope 		= SmartTags("Ver_Operador_Int_X")
   carga 		= SmartTags("Ver_Carga_X")
   programa 	= SmartTags("Ver_Programa_X")
   ciclovalido = SmartTags("Ver_CicloValido_X")
   
   'Crear consulta de insersion
   SQL_Table = "UPDATE Lav" & CStr(LavNro) & " SET fechafin = '" & CStr(fechafin)_
   		& "', fechainicio = '" 		& CStr(fechainicio)_
   		& "', cliente_0 = '" 		& CStr(cli1)_ 
   		& "', cliente_1 = '" 		& CStr(cli2)_
   		& "', cliente_2 = '" 		& CStr(cli3)_
   		& "', operario = '" 		& CStr(ope)_
   		& "', carga = '" 			& CStr(carga)_
   		& "', programa = '" 		& CStr(programa)_
   		& "', ciclovalido = '" 		& CStr(ciclovalido)_
   		& "' WHERE fechafin = '" 	& CStr(fechafin_ans) & "';"
   		
   
   Set rst302 = conn302.Execute(SQL_Table)
   
   'Error routine - Fehlerroutine
   If Err.Number <> 0 Then
   	bfde4b54-0db7-4817-8032-87127bf19bb9 "Error en ejecutar el update de base #" & Err.Number & " " & Err.Description
   	Err.Clear
   	Set conn302 = Nothing 
   	Exit Sub
   End If
   
   conn302.close
   
   Set rst302 = Nothing
   Set conn302 = Nothing
   
   bfde4b54-0db7-4817-8032-87127bf19bb9 "Salio a S401"

VB script "S402_ActRegDeEdicion"
   bfde4b54-0db7-4817-8032-87127bf19bb9 "Entro a S402"
   'Declaracion de Variables locales
   Dim connListLav, rstListLav, SQL_Table
   Dim Consulta, Dia
   On Error Resume Next
   
   Set connListLav = CreateObject("ADODB.Connection")
   'Abrir BDD
   connListLav.Open "Provider=MSDASQL;Initial Catalog=Lavadero;DSN=Lavadero"
   
   bfde4b54-0db7-4817-8032-87127bf19bb9 "Entro a S402_1"
   
   'Chequeo de error
   If Err.Number <> 0 Then
   	bfde4b54-0db7-4817-8032-87127bf19bb9 "Error al abrir BDD#" & Err.Number & " " & Err.Description
   	Err.Clear 
   	connListLav.close
   	Exit Sub
   End If
   
   'Dia que se esta visualizando
   Dia = SmartTags("Ver_DIA_X")
   
   	Consulta = "SELECT * FROM Lav" & CStr(LavNro) & " WHERE cast(fechafin as date) = '"
   	Consulta = Consulta & CStr(Year(Dia)) & "-" & CStr(Month(Dia)) & "-" & CStr(Day(Dia)) & "' "
   	Consulta = Consulta & "and cast(fechafin as time) like '%" & TimeSerial(Hour(SmartTags("Ver_HoraFin_" & CStr(RegNro))), Minute(SmartTags("Ver_HoraFin_" & CStr(RegNro))), Second(SmartTags("Ver_HoraFin_" & CStr(RegNro)))) & "%'"
   	
   	'Select * from Lav1 where cast(fechafin as Date) =  '2020-08-19' and cast(fechafin as time) like '%09:00:30%'
   	
   	bfde4b54-0db7-4817-8032-87127bf19bb9 "Entro a S402_2"
   Set rstListLav = CreateObject("ADODB.Recordset")
   'Ejecutar consulta
   Set rstListLav = connListLav.Execute(Consulta)
   
   If Err.Number <> 0 Then
   	bfde4b54-0db7-4817-8032-87127bf19bb9 "Error en Consulta S402_3 #" & Err.Number & " " & Err.Description
   	Err.Clear
   	rstListLav.close
   	connListLav.close 
   	'Exit Sub
   End If
   
   bfde4b54-0db7-4817-8032-87127bf19bb9 "Entro a S402_3"
   
   
   'Llenado de variables que muestan la lista
   	
   	If rstListLav.EOF = False Then
   		SmartTags("Ver_HoraFin_X_ans") 		= rstListLav.Fields(0).Value
   		SmartTags("Ver_HoraInicio_X_ans") 	= rstListLav.Fields(1).Value
   		SmartTags("Ver_Cli1_Str_X_ans")		= rstListLav.Fields(2).Value
   		SmartTags("Ver_Cli2_Str_X_ans")		= rstListLav.Fields(3).Value
   		SmartTags("Ver_Cli3_Str_X_ans")		= rstListLav.Fields(4).Value
   		SmartTags("Ver_Operador_Int_X_ans")	= rstListLav.Fields(5).Value
   		SmartTags("Ver_Carga_X_ans") 		= rstListLav.Fields(6).Value
   		SmartTags("Ver_Programa_X_ans")		= rstListLav.Fields(7).Value
   		SmartTags("Ver_CicloValido_X_ans")	= rstListLav.Fields(8).Value
   		
   		SmartTags("Ver_HoraFin_X") 		= SmartTags("Ver_HoraFin_X_ans")
   		SmartTags("Ver_HoraInicio_X") 	= SmartTags("Ver_HoraInicio_X_ans")
   		SmartTags("Ver_Cli1_Str_X")		= SmartTags("Ver_Cli1_Str_X_ans")
   		SmartTags("Ver_Cli2_Str_X")		= SmartTags("Ver_Cli2_Str_X_ans")
   		SmartTags("Ver_Cli3_Str_X")		= SmartTags("Ver_Cli3_Str_X_ans")
   		SmartTags("Ver_Operador_Int_X")	= SmartTags("Ver_Operador_Int_X_ans")
   		SmartTags("Ver_Carga_X") 		= SmartTags("Ver_Carga_X_ans")
   		SmartTags("Ver_Programa_X")		= SmartTags("Ver_Programa_X_ans")
   		SmartTags("Ver_CicloValido_X")	= SmartTags("Ver_CicloValido_X_ans")
   	End If
   	
   If Err.Number <> 0 Then
   	bfde4b54-0db7-4817-8032-87127bf19bb9 "Error en grabar los datos en variables" & Err.Number & " " & Err.Description
   	Err.Clear
   	rstListLav.close
   	connListLav.close 
   	'Exit Sub
   End If
   
   bfde4b54-0db7-4817-8032-87127bf19bb9 "Entro a S400_5"
   ''''''''''''''''''''''''''''''''''''''''''''''''''''''''''''''''''''''''''''''
   '########################################################################
   
   
   rstListLav.close
   connListLav.close
   
   Set rstListLav = Nothing
   Set connListLav = Nothing
   
   If Err.Number <> 0 Then
   	bfde4b54-0db7-4817-8032-87127bf19bb9 "Error en establecer los operadores#" & Err.Number & " " & Err.Description
   	Err.Clear
   	rstListLav.close
   	connListLav.close
   	Exit Sub
   End If
   
   bfde4b54-0db7-4817-8032-87127bf19bb9 "Salio a S402"

VB script "S500_InformePeriodico"
   On Error Resume Next
   bfde4b54-0db7-4817-8032-87127bf19bb9 "Entro a S500 - Informe Periodico, tipo: " & tipo_Inf
   'Declaration of local tags 
   
   Dim cantidadDeLavadoras
   	cantidadDeLavadoras = 4
   
   Dim conn, rst, i, j, indicehoja, k, l, VarPR, VarC
   
   Dim Consulta,where, mesdesde, meshasta, diadesde, diahasta
   
   Dim impDesde, impHasta, impTipo
   Dim tCargaBraun(15), tCargaGirbau(15), promedioTotal(15), programaBraun(15), programaGirbau(15)
   
   ' Creo Variables locales para poder iterar con los datos
   Dim LavadoraNro
   
   
   'Inicializacion Global de variables
   For i = 1 To 15
   	tCargaBraun(i) = 0
   	tCargaGirbau(i) = 0
   	promedioTotal(i) = 0
   	programaBraun(i) = 0
   	programaGirbau(i) = 0
   Next
   
   If Err.Number <> 0 Then
   	bfde4b54-0db7-4817-8032-87127bf19bb9 "Consulta S500 Error 1#" & Err.Number & " " & Err.Description
   	Err.Clear
   	'Close data source
   	Set conn = Nothing
   	Set rst = Nothing 
   	
   	Exit Sub
   End If
   
   
   Select Case tipo_Inf
   	Case 0 ' Periodico
   		
   		If Month(desde) < 10 Then
   			mesdesde = "0" + CStr(Month(desde))
   		Else
   			mesdesde = CStr(Month(desde))
   		End If
   		
   		If Month(hasta) < 10 Then
   			meshasta = "0" + CStr(Month(hasta))
   		Else
   			meshasta = CStr(Month(hasta))
   		End If
   		
   		If Day(desde) < 10 Then
   			diadesde = "0" + CStr(Day(desde))
   		Else
   			diadesde = CStr(Day(desde))
   		End If
   		
   		If Day(hasta) < 10 Then
   			diahasta = "0" + CStr(Day(hasta))
   		Else
   			diahasta = CStr(Day(hasta))
   		End If
   		
   		
   				
   		where =" WHERE cast(fechafin As Date) >= '"
   		where = where & CStr(Year(desde)) & "-" & mesdesde & "-" & diadesde & "' "
   		where = where & "and cast(fechafin As Date) <= '"
   		where = where & CStr(Year(hasta)) & "-" & meshasta & "-" & diahasta & "' "
   		where = where & " order by fechafin"
   		
   		impDesde = CStr(Year(desde)) & "-" & mesdesde & "-" & diadesde
   		impHasta = CStr(Year(hasta)) & "-" & meshasta & "-" & diahasta
   		impTipo = "Periodico"
   		
   	Case 1 'Mensual
   		If hasta < 10 Then
   			meshasta = "0" + CStr(hasta)
   		Else
   			meshasta = CStr(hasta)
   		End If
   			
   		desde = Year(Date())
   		
   		
   		where = " WHERE cast(fechafin As Date) like '%"
   		where = where & CStr(desde) & "-" & meshasta & "%' "
   		where = where & "order by fechafin"
   		
   		impDesde = CStr(desde) & "-" & meshasta & "-01"
   		impHasta = CStr(desde) & "-" & meshasta & "-" & CStr(S406_UltimoDiaDelMes(meshasta,desde))
   		impTipo = "Mensual"
   		
   	Case 2 'Anual
   		
   		where = " WHERE cast(fechafin As Date) like '%"
   		where = where & CStr(hasta) & "-%' "
   		where = where & "order by fechafin"
   		
   		impDesde = CStr(hasta) & "-01-01"
   		impHasta = CStr(hasta) & "-12-31"
   		impTipo = "Anual"
   		
   End Select
   
   If Err.Number <> 0 Then
   	bfde4b54-0db7-4817-8032-87127bf19bb9 "Consulta Lav Error 3#" & Err.Number & " " & Err.Description
   	Err.Clear
   	'Close data source
   	Set conn = Nothing
   	Set rst = Nothing 
   	Exit Sub
   End If
   
   ' Comienzo de procesamiento de datos
   
   For LavadoraNro = 1 To cantidadDeLavadoras
   	'""""""""""""""""""""""""""""""""""""""""""""""""""""""""""""""""""""""""""""""""""""
   	' #################   Generacion de consulta a BDD Lavadora   ######################
   	'------------------------------------------------------------------------------------
   	'############ Estructura de datos de la Tabla Lav1 #################################
   	
   	'0			1			2			3			4			5			6			7			8			
   	'|FechaFin	|FechIni	|Cliente_0	|Cliente_1	|Cliente_2	|Operario	|Carga		|Programa	|Valido
   	'|Date		|Date		|Int		|Int		|Int		|Int		|Int 100g	|Int		|Bool
   	
   	'##################################################################################
   		
   	'''''''''''''''''''''''''''''''''''''''''''''''''''''''''''''''''''''''''''''
   	' #################   Procesamieno de Datos   #############################
   	'----------------------------------------------------------------------------
   	
   	'Ejecutar consulta
   	
   	Consulta = "SELECT * FROM Lav" & LavadoraNro & where
   	bfde4b54-0db7-4817-8032-87127bf19bb9 "Consulta " & Consulta
   			
   	
   	Set conn = CreateObject("ADODB.Connection")
   	conn.Open "Provider=MSDASQL;Initial Catalog=Lavadero;DSN=Lavadero"
   	Set rst = CreateObject("ADODB.Recordset")
   	Set rst = conn.Execute(Consulta)	
   		If Err.Number <> 0 Then
   			bfde4b54-0db7-4817-8032-87127bf19bb9 "Error en S500 - en la asignacion de variables ejecucion consulta en loop#" & Err.Number & " " & Err.Description
   			Err.Clear
   			Set conn = Nothing  
   			Exit Sub
   		End If
   
   	bfde4b54-0db7-4817-8032-87127bf19bb9 "Entra al loop de Lectura de registros de S500, lav nro " & LavadoraNro
   	
   	Do While rst.EOF = False
   		
